  MoveC 5273 to (-170.79, 260.24, -44.5) mm, rotated rx -180 ry 0 rz 0.01 deg; joints [38.208, -42.51, 99.953, -137.192, 65.567, 159.929] to (-173.38, 259.8, -44.5) mm, rotated rx -180 ry 0 rz 0.01 deg; joints [38.136, -42.43, 99.783, -137.238, 65.475, 159.893]
  MoveC 5274 to (-175.99, 259.57, -44.5) mm, rotated rx 180 ry 0 rz 0.01 deg; joints [38.069, -42.344, 99.599, -137.276, 65.378, 159.849] to (-178.62, 259.49, -44.5) mm, rotated rx 180 ry 0 rz 0.01 deg; joints [38.007, -42.253, 99.403, -137.307, 65.279, 159.798]
  MoveL 5275 to (-216.35, 259.58, -44.5) mm, rotated rx 180 ry 0 rz 0.01 deg; joints [37.165, -40.878, 96.467, -137.67, 63.812, 159.01]
  MoveC 5276 to (-223.68, 260.93, -44.5) mm, rotated rx 180 ry 0 rz 0.01 deg; joints [37.043, -40.567, 95.803, -137.677, 63.505, 158.802] to (-230.83, 263.03, -44.5) mm, rotated rx 180 ry 0 rz 0.01 deg; joints [36.949, -40.24, 95.104, -137.649, 63.193, 158.566]
  MoveC 5277 to (-237.52, 266.44, -44.5) mm, rotated rx -180 ry 0 rz 0.01 deg; joints [36.902, -39.891, 94.357, -137.561, 62.881, 158.288] to (-243.08, 271.47, -44.5) mm, rotated rx -180 ry 0 rz 0.01 deg; joints [36.926, -39.537, 93.597, -137.394, 62.592, 157.967]
  MoveC 5278 to (-246.21, 275.5, -44.5) mm, rotated rx 180 ry 0 rz 0.01 deg; joints [36.974, -39.303, 93.093, -137.25, 62.413, 157.738] to (-248.99, 279.78, -44.5) mm, rotated rx 180 ry 0 rz 0.01 deg; joints [37.036, -39.073, 92.601, -137.092, 62.245, 157.506]
  MoveC 5279 to (-251.23, 284.38, -44.5) mm, rotated rx 180 ry 0 rz 0.01 deg; joints [37.118, -38.854, 92.13, -136.916, 62.094, 157.271] to (-252.73, 289.26, -44.5) mm, rotated rx -180 ry 0 rz 0.01 deg; joints [37.224, -38.654, 91.699, -136.724, 61.969, 157.04]
  MoveC 5280 to (-253.82, 296.03, -44.5) mm, rotated rx -180 ry 0 rz 0.01 deg; joints [37.39, -38.415, 91.182, -136.45, 61.836, 156.741] to (-254.09, 302.88, -44.5) mm, rotated rx 180 ry 0 rz 0.01 deg; joints [37.576, -38.202, 90.723, -136.168, 61.736, 156.455]
  MoveC 5281 to (-253.11, 309.7, -44.5) mm, rotated rx -180 ry 0 rz 0.01 deg; joints [37.786, -38.038, 90.366, -135.879, 61.686, 156.199] to (-250.53, 316.09, -44.5) mm, rotated rx -180 ry 0 rz 0.01 deg; joints [38.018, -37.948, 90.167, -135.6, 61.707, 155.997]
  MoveC 5282 to (-249.34, 318.22, -44.5) mm, rotated rx -180 ry 0 rz 0.01 deg; joints [38.102, -37.931, 90.127, -135.505, 61.727, 155.937] to (-248.13, 320.34, -44.5) mm, rotated rx 180 ry 0 rz 0.01 deg; joints [38.187, -37.915, 90.089, -135.41, 61.748, 155.878]
  MoveL 5283 to (-247.97, 320.95, -44.33) mm, rotated rx 180 ry 0 rz 0.01 deg; joints [38.207, -37.911, 90.064, -135.382, 61.741, 155.851]
  MoveL 5284 to (-248.05, 321.41, -43.87) mm, rotated rx -180 ry 0 rz 0.01 deg; joints [38.217, -37.915, 90.03, -135.356, 61.718, 155.815]
  MoveL 5285 to (-248.12, 321.56, -43.23) mm, rotated rx 180 ry 0 rz 0.01 deg; joints [38.22, -37.938, 90.017, -135.34, 61.694, 155.785]
  Set speed (500.0 mm/s)
  MoveL 5286 to (-248.12, 321.56, 11) mm, rotated rx -180 ry 0 rz 0.01 deg; joints [38.197, -40.432, 90.187, -134.447, 60.044, 153.913]
  Set speed (500.0 mm/s)
  MoveL 5287 to (-399.69, 339.08, 11) mm, rotated rx 180 ry 0 rz 0.01 deg; joints [35.607, -32.97, 75.014, -133.485, 53.388, 148.774]
  Set speed (100.0 mm/s)
  MoveL 5288 to (-399.69, 339.08, -28.23) mm, rotated rx -180 ry 0 rz 0.01 deg; joints [35.623, -31.334, 74.905, -134.27, 54.456, 150.126]
  MoveL 5289 to (-399.69, 339.08, -28.33) mm, rotated rx -180 ry 0 rz 0.01 deg; joints [35.623, -31.33, 74.904, -134.272, 54.458, 150.13]
  MoveL 5290 to (-399.83, 339.05, -28.81) mm, rotated rx -180 ry 0 rz 0.01 deg; joints [35.62, -31.303, 74.89, -134.281, 54.465, 150.142]
  MoveL 5291 to (-400.13, 338.98, -29.2) mm, rotated rx -180 ry 0 rz 0.01 deg; joints [35.613, -31.274, 74.862, -134.289, 54.462, 150.148]
  MoveL 5292 to (-400.55, 338.85, -29.44) mm, rotated rx -180 ry 0 rz 0.01 deg; joints [35.602, -31.247, 74.827, -134.297, 54.45, 150.148]
  MoveL 5293 to (-400.6, 338.83, -29.46) mm, rotated rx -180 ry 0 rz 0.01 deg; joints [35.6, -31.245, 74.824, -134.298, 54.449, 150.148]
  MoveL 5294 to (-400.86, 338.72, -29.5) mm, rotated rx 180 ry 0 rz 0.01 deg; joints [35.593, -31.234, 74.805, -134.302, 54.439, 150.145]
  MoveL 5295 to (-401.28, 338.49, -29.52) mm, rotated rx 180 ry 0 rz 0.01 deg; joints [35.579, -31.22, 74.778, -134.31, 54.423, 150.143]
  MoveL 5296 to (-401.4, 338.42, -29.52) mm, rotated rx 180 ry 0 rz 0.01 deg; joints [35.574, -31.216, 74.771, -134.313, 54.418, 150.142]
  MoveL 5297 to (-402.84, 337.05, -29.59) mm, rotated rx 180 ry 0 rz 0.01 deg; joints [35.511, -31.189, 74.722, -134.368, 54.371, 150.163]
  MoveL 5298 to (-402.87, 337.02, -29.59) mm, rotated rx -180 ry 0 rz 0.01 deg; joints [35.51, -31.189, 74.722, -134.37, 54.37, 150.164]
  MoveL 5299 to (-403.75, 334.43, -29.69) mm, rotated rx -180 ry 0 rz 0.01 deg; joints [35.425, -31.231, 74.821, -134.488, 54.366, 150.266]
  MoveL 5300 to (-403.78, 333.95, -29.71) mm, rotated rx -180 ry 0 rz 0.01 deg; joints [35.412, -31.246, 74.854, -134.511, 54.372, 150.29]
  MoveL 5301 to (-403.79, 333.65, -29.72) mm, rotated rx -180 ry 0 rz 0.01 deg; joints [35.404, -31.255, 74.874, -134.525, 54.375, 150.305]
  MoveL 5302 to (-403.79, 333.05, -29.74) mm, rotated rx -180 ry 0 rz 0.01 deg; joints [35.388, -31.276, 74.919, -134.554, 54.384, 150.336]
  MoveL 5303 to (-401.25, 328.08, -29.94) mm, rotated rx -180 ry 0 rz 0.01 deg; joints [35.304, -31.566, 75.542, -134.812, 54.575, 150.679]
  MoveL 5304 to (-395.74, 327.2, -30.14) mm, rotated rx -180 ry 0 rz 0.01 deg; joints [35.385, -31.86, 76.168, -134.893, 54.85, 150.918]
  MoveL 5305 to (-391.79, 331.15, -30.35) mm, rotated rx -180 ry 0 rz 0.01 deg; joints [35.564, -31.91, 76.283, -134.736, 54.987, 150.863]
  MoveL 5306 to (-392.66, 336.66, -30.55) mm, rotated rx -180 ry 0 rz 0.01 deg; joints [35.694, -31.668, 75.792, -134.476, 54.878, 150.567]
  MoveL 5307 to (-397.64, 339.2, -30.75) mm, rotated rx -180 ry 0 rz 0.01 deg; joints [35.666, -31.325, 75.096, -134.327, 54.617, 150.275]
  MoveL 5308 to (-398.51, 339.2, -30.78) mm, rotated rx -180 ry 0 rz 0.01 deg; joints [35.65, -31.28, 75.006, -134.321, 54.577, 150.246]
  MoveL 5309 to (-399.34, 339.13, -30.81) mm, rotated rx 180 ry 0 rz 0.01 deg; joints [35.633, -31.24, 74.926, -134.319, 54.54, 150.221]
  MoveL 5310 to (-399.69, 339.08, -30.82) mm, rotated rx -180 ry 0 rz 0.01 deg; joints [35.624, -31.223, 74.893, -134.319, 54.525, 150.212]
  MoveL 5311 to (-400.55, 338.85, -30.85) mm, rotated rx -180 ry 0 rz 0.01 deg; joints [35.602, -31.187, 74.821, -134.324, 54.488, 150.194]
  MoveL 5312 to (-400.6, 338.83, -30.85) mm, rotated rx -180 ry 0 rz 0.01 deg; joints [35.601, -31.185, 74.818, -134.324, 54.486, 150.194]
  MoveL 5313 to (-401.28, 338.49, -30.88) mm, rotated rx -180 ry 0 rz 0.01 deg; joints [35.579, -31.162, 74.772, -134.336, 54.459, 150.188]
  MoveL 5314 to (-401.4, 338.42, -30.89) mm, rotated rx -180 ry 0 rz 0.01 deg; joints [35.575, -31.158, 74.764, -134.339, 54.455, 150.187]
  MoveL 5315 to (-402.84, 337.05, -30.96) mm, rotated rx -180 ry 0 rz 0.01 deg; joints [35.512, -31.131, 74.716, -134.394, 54.407, 150.208]
  MoveL 5316 to (-402.87, 337.02, -30.96) mm, rotated rx -180 ry 0 rz 0.01 deg; joints [35.511, -31.131, 74.716, -134.395, 54.407, 150.209]
  MoveL 5317 to (-403.75, 334.43, -31.05) mm, rotated rx 180 ry 0 rz 0.01 deg; joints [35.426, -31.173, 74.814, -134.514, 54.402, 150.311]
  MoveL 5318 to (-403.78, 333.95, -31.07) mm, rotated rx -180 ry 0 rz 0.01 deg; joints [35.413, -31.188, 74.847, -134.537, 54.408, 150.335]
  MoveL 5319 to (-403.79, 333.65, -31.08) mm, rotated rx 180 ry 0 rz 0.01 deg; joints [35.405, -31.197, 74.868, -134.551, 54.412, 150.35]
  MoveL 5320 to (-403.79, 333.05, -31.1) mm, rotated rx 180 ry 0 rz 0.01 deg; joints [35.389, -31.217, 74.912, -134.58, 54.421, 150.381]
  MoveL 5321 to (-401.25, 328.08, -31.3) mm, rotated rx -180 ry 0 rz 0.01 deg; joints [35.305, -31.508, 75.536, -134.837, 54.612, 150.724]
  MoveL 5322 to (-395.74, 327.2, -31.51) mm, rotated rx 180 ry 0 rz 0.01 deg; joints [35.386, -31.801, 76.162, -134.918, 54.888, 150.962]
  MoveL 5323 to (-391.79, 331.15, -31.71) mm, rotated rx 180 ry 0 rz 0.01 deg; joints [35.565, -31.851, 76.276, -134.762, 55.024, 150.908]
  MoveL 5324 to (-392.66, 336.66, -31.91) mm, rotated rx 180 ry 0 rz 0.01 deg; joints [35.694, -31.609, 75.785, -134.502, 54.915, 150.612]
  MoveL 5325 to (-397.64, 339.2, -32.11) mm, rotated rx -180 ry 0 rz 0.01 deg; joints [35.667, -31.266, 75.089, -134.352, 54.654, 150.32]
  MoveL 5326 to (-398.51, 339.2, -32.14) mm, rotated rx -180 ry 0 rz 0.01 deg; joints [35.651, -31.222, 75, -134.347, 54.614, 150.291]
  MoveL 5327 to (-399.34, 339.13, -32.17) mm, rotated rx -180 ry 0 rz 0.01 deg; joints [35.633, -31.181, 74.919, -134.344, 54.577, 150.266]
  MoveL 5328 to (-399.69, 339.08, -32.19) mm, rotated rx 180 ry 0 rz 0.01 deg; joints [35.625, -31.165, 74.886, -134.345, 54.561, 150.257]
  MoveL 5329 to (-400.55, 338.85, -32.22) mm, rotated rx 180 ry 0 rz 0.01 deg; joints [35.603, -31.129, 74.814, -134.35, 54.525, 150.239]
  MoveL 5330 to (-400.6, 338.83, -32.22) mm, rotated rx -180 ry 0 rz 0.01 deg; joints [35.602, -31.127, 74.811, -134.35, 54.523, 150.239]
  MoveL 5331 to (-401.28, 338.49, -32.25) mm, rotated rx 180 ry 0 rz 0.01 deg; joints [35.58, -31.104, 74.765, -134.362, 54.496, 150.233]
  MoveL 5332 to (-401.4, 338.42, -32.25) mm, rotated rx -180 ry 0 rz 0.01 deg; joints [35.575, -31.1, 74.758, -134.364, 54.491, 150.232]
  MoveL 5333 to (-402.84, 337.05, -32.32) mm, rotated rx -180 ry 0 rz 0.01 deg; joints [35.513, -31.073, 74.709, -134.42, 54.444, 150.253]
  MoveL 5334 to (-402.87, 337.02, -32.32) mm, rotated rx -180 ry 0 rz 0.01 deg; joints [35.511, -31.073, 74.709, -134.421, 54.443, 150.254]
  MoveL 5335 to (-403.75, 334.43, -32.42) mm, rotated rx -180 ry 0 rz 0.01 deg; joints [35.426, -31.115, 74.808, -134.539, 54.439, 150.356]
  MoveL 5336 to (-403.78, 333.95, -32.44) mm, rotated rx -180 ry 0 rz 0.01 deg; joints [35.413, -31.13, 74.841, -134.562, 54.445, 150.38]
  MoveL 5337 to (-403.79, 333.65, -32.45) mm, rotated rx -180 ry 0 rz 0.01 deg; joints [35.405, -31.139, 74.861, -134.576, 54.449, 150.395]
  MoveL 5338 to (-403.79, 333.05, -32.47) mm, rotated rx -180 ry 0 rz 0.01 deg; joints [35.389, -31.159, 74.906, -134.605, 54.457, 150.426]
  MoveL 5339 to (-401.25, 328.08, -32.67) mm, rotated rx -180 ry 0 rz 0.01 deg; joints [35.306, -31.449, 75.529, -134.863, 54.649, 150.769]
  MoveL 5340 to (-395.74, 327.2, -32.87) mm, rotated rx 180 ry 0 rz 0.01 deg; joints [35.386, -31.743, 76.155, -134.944, 54.925, 151.007]
  MoveL 5341 to (-391.79, 331.15, -33.07) mm, rotated rx -180 ry 0 rz 0.01 deg; joints [35.565, -31.793, 76.27, -134.787, 55.061, 150.953]
  MoveL 5342 to (-392.66, 336.66, -33.28) mm, rotated rx -180 ry 0 rz 0.01 deg; joints [35.695, -31.551, 75.779, -134.527, 54.952, 150.657]
  MoveL 5343 to (-397.64, 339.2, -33.48) mm, rotated rx -180 ry 0 rz 0.01 deg; joints [35.668, -31.208, 75.083, -134.378, 54.69, 150.365]
  MoveL 5344 to (-398.51, 339.2, -33.51) mm, rotated rx -180 ry 0 rz 0.01 deg; joints [35.651, -31.163, 74.993, -134.372, 54.65, 150.336]
  MoveL 5345 to (-399.34, 339.13, -33.54) mm, rotated rx -180 ry 0 rz 0.01 deg; joints [35.634, -31.123, 74.912, -134.37, 54.613, 150.311]
  MoveL 5346 to (-399.69, 339.08, -33.55) mm, rotated rx -180 ry 0 rz 0.01 deg; joints [35.626, -31.107, 74.88, -134.37, 54.597, 150.302]
  MoveL 5347 to (-400.55, 338.85, -33.58) mm, rotated rx -180 ry 0 rz 0.01 deg; joints [35.603, -31.071, 74.807, -134.375, 54.561, 150.284]
  MoveL 5348 to (-400.6, 338.83, -33.58) mm, rotated rx -180 ry 0 rz 0.01 deg; joints [35.602, -31.069, 74.804, -134.376, 54.559, 150.284]
  MoveL 5349 to (-401.28, 338.49, -33.61) mm, rotated rx -180 ry 0 rz 0.01 deg; joints [35.58, -31.045, 74.758, -134.387, 54.532, 150.278]
  MoveL 5350 to (-401.4, 338.42, -33.62) mm, rotated rx -180 ry 0 rz 0.01 deg; joints [35.576, -31.042, 74.751, -134.39, 54.527, 150.277]
  MoveL 5351 to (-402.84, 337.05, -33.69) mm, rotated rx 180 ry 0 rz 0.01 deg; joints [35.513, -31.015, 74.703, -134.445, 54.48, 150.298]
  MoveL 5352 to (-402.87, 337.02, -33.69) mm, rotated rx -180 ry 0 rz 0.01 deg; joints [35.512, -31.015, 74.703, -134.447, 54.479, 150.299]
  MoveL 5353 to (-403.75, 334.43, -33.78) mm, rotated rx -180 ry 0 rz 0.01 deg; joints [35.427, -31.056, 74.801, -134.565, 54.475, 150.401]
  MoveL 5354 to (-403.78, 333.95, -33.8) mm, rotated rx 180 ry 0 rz 0.01 deg; joints [35.414, -31.071, 74.834, -134.588, 54.481, 150.425]
  MoveL 5355 to (-403.79, 333.65, -33.81) mm, rotated rx -180 ry 0 rz 0.01 deg; joints [35.406, -31.081, 74.855, -134.602, 54.485, 150.44]
  MoveL 5356 to (-403.79, 333.05, -33.83) mm, rotated rx -180 ry 0 rz 0.01 deg; joints [35.39, -31.101, 74.899, -134.631, 54.494, 150.471]
  MoveL 5357 to (-401.25, 328.08, -34.03) mm, rotated rx 180 ry 0 rz 0.01 deg; joints [35.306, -31.391, 75.523, -134.888, 54.686, 150.814]
  MoveL 5358 to (-395.74, 327.2, -34.24) mm, rotated rx -180 ry 0 rz 0.01 deg; joints [35.387, -31.684, 76.148, -134.969, 54.962, 151.052]
  MoveL 5359 to (-391.79, 331.15, -34.44) mm, rotated rx -180 ry 0 rz 0.01 deg; joints [35.566, -31.734, 76.263, -134.812, 55.098, 150.998]
  MoveL 5360 to (-392.66, 336.66, -34.64) mm, rotated rx -180 ry 0 rz 0.01 deg; joints [35.695, -31.492, 75.772, -134.552, 54.988, 150.702]
  MoveL 5361 to (-397.64, 339.2, -34.84) mm, rotated rx -180 ry 0 rz 0.01 deg; joints [35.668, -31.149, 75.076, -134.403, 54.727, 150.41]
  MoveL 5362 to (-398.51, 339.2, -34.87) mm, rotated rx 180 ry 0 rz 0.01 deg; joints [35.652, -31.105, 74.986, -134.398, 54.687, 150.381]
  MoveL 5363 to (-399.34, 339.13, -34.9) mm, rotated rx -180 ry 0 rz 0.01 deg; joints [35.634, -31.065, 74.905, -134.395, 54.649, 150.356]
  MoveL 5364 to (-399.69, 339.08, -34.92) mm, rotated rx -180 ry 0 rz 0.01 deg; joints [35.626, -31.048, 74.873, -134.396, 54.634, 150.347]
  MoveL 5365 to (-400.55, 338.85, -34.95) mm, rotated rx -180 ry 0 rz 0.01 deg; joints [35.604, -31.012, 74.801, -134.401, 54.597, 150.329]
  MoveL 5366 to (-400.6, 338.83, -34.95) mm, rotated rx -180 ry 0 rz 0.01 deg; joints [35.603, -31.011, 74.797, -134.401, 54.595, 150.329]
  MoveL 5367 to (-401.28, 338.49, -34.97) mm, rotated rx 180 ry 0 rz 0.01 deg; joints [35.581, -30.987, 74.751, -134.413, 54.568, 150.322]
  MoveL 5368 to (-401.4, 338.42, -34.98) mm, rotated rx -180 ry 0 rz 0.01 deg; joints [35.577, -30.983, 74.744, -134.416, 54.564, 150.322]
  MoveL 5369 to (-402.84, 337.05, -35.05) mm, rotated rx -180 ry 0 rz 0.01 deg; joints [35.514, -30.956, 74.696, -134.471, 54.516, 150.342]
  MoveL 5370 to (-402.87, 337.02, -35.05) mm, rotated rx -180 ry 0 rz 0.01 deg; joints [35.512, -30.956, 74.696, -134.472, 54.516, 150.343]
  MoveL 5371 to (-403.75, 334.43, -35.15) mm, rotated rx -180 ry 0 rz 0.01 deg; joints [35.428, -30.998, 74.794, -134.59, 54.512, 150.445]
  MoveL 5372 to (-403.78, 333.95, -35.16) mm, rotated rx 180 ry 0 rz 0.01 deg; joints [35.414, -31.013, 74.827, -134.613, 54.518, 150.469]
  MoveL 5373 to (-403.79, 333.65, -35.18) mm, rotated rx 180 ry 0 rz 0.01 deg; joints [35.406, -31.022, 74.848, -134.628, 54.521, 150.484]
  MoveL 5374 to (-403.79, 333.05, -35.2) mm, rotated rx -180 ry 0 rz 0.01 deg; joints [35.391, -31.042, 74.892, -134.657, 54.53, 150.515]
  MoveL 5375 to (-401.25, 328.08, -35.4) mm, rotated rx -180 ry 0 rz 0.01 deg; joints [35.307, -31.332, 75.516, -134.913, 54.723, 150.858]
  MoveL 5376 to (-395.74, 327.2, -35.6) mm, rotated rx -180 ry 0 rz 0.01 deg; joints [35.387, -31.625, 76.141, -134.994, 54.999, 151.096]
  MoveL 5377 to (-391.79, 331.15, -35.8) mm, rotated rx -180 ry 0 rz 0.01 deg; joints [35.567, -31.675, 76.256, -134.837, 55.135, 151.042]
  MoveL 5378 to (-392.66, 336.66, -36.01) mm, rotated rx -180 ry 0 rz 0.01 deg; joints [35.696, -31.434, 75.765, -134.577, 55.025, 150.747]
  MoveL 5379 to (-397.64, 339.2, -36.21) mm, rotated rx 180 ry 0 rz 0.01 deg; joints [35.669, -31.091, 75.069, -134.429, 54.763, 150.455]
  MoveL 5380 to (-398.51, 339.2, -36.24) mm, rotated rx -180 ry 0 rz 0.01 deg; joints [35.652, -31.046, 74.979, -134.423, 54.723, 150.426]
  MoveL 5381 to (-399.34, 339.13, -36.27) mm, rotated rx 180 ry 0 rz 0.01 deg; joints [35.635, -31.006, 74.898, -134.421, 54.686, 150.401]
  MoveL 5382 to (-399.69, 339.08, -36.28) mm, rotated rx 180 ry 0 rz 0.01 deg; joints [35.627, -30.99, 74.866, -134.421, 54.67, 150.392]
  MoveL 5383 to (-400.55, 338.85, -36.31) mm, rotated rx 180 ry 0 rz 0.01 deg; joints [35.605, -30.954, 74.793, -134.426, 54.633, 150.374]
  MoveL 5384 to (-400.6, 338.83, -36.31) mm, rotated rx 180 ry 0 rz 0.01 deg; joints [35.603, -30.952, 74.79, -134.427, 54.632, 150.373]
  MoveL 5385 to (-401.28, 338.49, -36.34) mm, rotated rx -180 ry 0 rz 0.01 deg; joints [35.582, -30.929, 74.744, -134.438, 54.605, 150.367]
  MoveL 5386 to (-401.4, 338.42, -36.34) mm, rotated rx -180 ry 0 rz 0.01 deg; joints [35.577, -30.925, 74.737, -134.441, 54.6, 150.367]
  MoveL 5387 to (-402.84, 337.05, -36.41) mm, rotated rx -180 ry 0 rz 0.01 deg; joints [35.514, -30.898, 74.689, -134.496, 54.553, 150.387]
  MoveL 5388 to (-402.87, 337.02, -36.42) mm, rotated rx -180 ry 0 rz 0.01 deg; joints [35.513, -30.898, 74.689, -134.498, 54.552, 150.388]
  MoveL 5389 to (-403.75, 334.43, -36.51) mm, rotated rx -180 ry 0 rz 0.01 deg; joints [35.428, -30.94, 74.787, -134.616, 54.548, 150.49]
  MoveL 5390 to (-403.78, 333.95, -36.53) mm, rotated rx -180 ry 0 rz 0.01 deg; joints [35.415, -30.954, 74.82, -134.639, 54.554, 150.514]
  MoveL 5391 to (-403.79, 333.65, -36.54) mm, rotated rx -180 ry 0 rz 0.01 deg; joints [35.407, -30.964, 74.841, -134.653, 54.558, 150.529]
  MoveL 5392 to (-403.79, 333.05, -36.56) mm, rotated rx -180 ry 0 rz 0.01 deg; joints [35.391, -30.984, 74.885, -134.682, 54.567, 150.56]
  MoveL 5393 to (-401.25, 328.08, -36.76) mm, rotated rx 180 ry 0 rz 0.01 deg; joints [35.307, -31.273, 75.509, -134.938, 54.759, 150.902]
  MoveL 5394 to (-395.74, 327.2, -36.97) mm, rotated rx -180 ry 0 rz 0.01 deg; joints [35.388, -31.566, 76.134, -135.019, 55.036, 151.14]
  MoveL 5395 to (-391.79, 331.15, -37.17) mm, rotated rx -180 ry 0 rz 0.01 deg; joints [35.567, -31.616, 76.249, -134.862, 55.172, 151.086]
  MoveL 5396 to (-392.66, 336.66, -37.37) mm, rotated rx 180 ry 0 rz 0.01 deg; joints [35.697, -31.375, 75.758, -134.603, 55.061, 150.791]
  MoveL 5397 to (-397.64, 339.2, -37.57) mm, rotated rx -180 ry 0 rz 0.01 deg; joints [35.669, -31.032, 75.061, -134.454, 54.799, 150.499]
  MoveL 5398 to (-398.51, 339.2, -37.6) mm, rotated rx 180 ry 0 rz 0.01 deg; joints [35.653, -30.988, 74.972, -134.448, 54.759, 150.47]
  MoveL 5399 to (-399.34, 339.13, -37.63) mm, rotated rx -180 ry 0 rz 0.01 deg; joints [35.636, -30.948, 74.891, -134.446, 54.722, 150.445]
  MoveL 5400 to (-399.69, 339.08, -37.64) mm, rotated rx 180 ry 0 rz 0.01 deg; joints [35.627, -30.931, 74.858, -134.447, 54.706, 150.436]
  MoveL 5401 to (-400.55, 338.85, -37.68) mm, rotated rx 180 ry 0 rz 0.01 deg; joints [35.605, -30.895, 74.786, -134.452, 54.67, 150.418]
  MoveL 5402 to (-400.6, 338.83, -37.68) mm, rotated rx -180 ry 0 rz 0.01 deg; joints [35.604, -30.894, 74.783, -134.452, 54.668, 150.418]
  MoveL 5403 to (-401.28, 338.49, -37.7) mm, rotated rx 180 ry 0 rz 0.01 deg; joints [35.582, -30.87, 74.737, -134.464, 54.641, 150.411]
  MoveL 5404 to (-401.4, 338.42, -37.71) mm, rotated rx -180 ry 0 rz 0.01 deg; joints [35.578, -30.866, 74.73, -134.466, 54.636, 150.411]
  MoveL 5405 to (-402.84, 337.05, -37.78) mm, rotated rx -180 ry 0 rz 0.01 deg; joints [35.515, -30.839, 74.681, -134.522, 54.589, 150.431]
  MoveL 5406 to (-402.87, 337.02, -37.78) mm, rotated rx -180 ry 0 rz 0.01 deg; joints [35.514, -30.839, 74.681, -134.523, 54.588, 150.432]
  MoveL 5407 to (-403.75, 334.43, -37.88) mm, rotated rx -180 ry 0 rz 0.01 deg; joints [35.429, -30.881, 74.78, -134.641, 54.584, 150.534]
  MoveL 5408 to (-403.78, 333.95, -37.89) mm, rotated rx -180 ry 0 rz 0.01 deg; joints [35.416, -30.896, 74.813, -134.664, 54.59, 150.558]
  MoveL 5409 to (-403.79, 333.65, -37.9) mm, rotated rx 180 ry 0 rz 0.01 deg; joints [35.408, -30.905, 74.833, -134.678, 54.594, 150.573]
  MoveL 5410 to (-403.79, 333.05, -37.93) mm, rotated rx -180 ry 0 rz 0.01 deg; joints [35.392, -30.925, 74.878, -134.707, 54.603, 150.604]
  MoveL 5411 to (-401.25, 328.08, -38.13) mm, rotated rx -180 ry 0 rz 0.01 deg; joints [35.308, -31.215, 75.501, -134.964, 54.796, 150.947]
  MoveL 5412 to (-395.74, 327.2, -38.33) mm, rotated rx -180 ry 0 rz 0.01 deg; joints [35.389, -31.507, 76.127, -135.044, 55.072, 151.185]
  MoveL 5413 to (-391.79, 331.15, -38.53) mm, rotated rx 180 ry 0 rz 0.01 deg; joints [35.568, -31.557, 76.242, -134.887, 55.209, 151.131]
  MoveL 5414 to (-392.66, 336.66, -38.73) mm, rotated rx 180 ry 0 rz 0.01 deg; joints [35.697, -31.316, 75.751, -134.628, 55.098, 150.835]
  MoveL 5415 to (-397.64, 339.2, -38.94) mm, rotated rx 180 ry 0 rz 0.01 deg; joints [35.67, -30.974, 75.054, -134.479, 54.835, 150.544]
  MoveL 5416 to (-398.51, 339.2, -38.97) mm, rotated rx -180 ry 0 rz 0.01 deg; joints [35.654, -30.929, 74.964, -134.474, 54.795, 150.514]
  MoveL 5417 to (-399.34, 339.13, -39) mm, rotated rx 180 ry 0 rz 0.01 deg; joints [35.636, -30.889, 74.884, -134.471, 54.758, 150.49]
  MoveL 5418 to (-399.69, 339.08, -39.01) mm, rotated rx -180 ry 0 rz 0.01 deg; joints [35.628, -30.873, 74.851, -134.472, 54.742, 150.48]
  MoveL 5419 to (-400.55, 338.85, -39.04) mm, rotated rx -180 ry 0 rz 0.01 deg; joints [35.606, -30.837, 74.779, -134.477, 54.706, 150.463]
  MoveL 5420 to (-400.6, 338.83, -39.04) mm, rotated rx 180 ry 0 rz 0.01 deg; joints [35.605, -30.835, 74.776, -134.477, 54.704, 150.462]
  MoveL 5421 to (-401.28, 338.49, -39.07) mm, rotated rx 180 ry 0 rz 0.01 deg; joints [35.583, -30.811, 74.73, -134.489, 54.677, 150.456]
  MoveL 5422 to (-401.4, 338.42, -39.07) mm, rotated rx 180 ry 0 rz 0.01 deg; joints [35.578, -30.808, 74.722, -134.492, 54.672, 150.456]
  MoveL 5423 to (-402.84, 337.05, -39.14) mm, rotated rx 180 ry 0 rz 0.01 deg; joints [35.516, -30.781, 74.674, -134.547, 54.625, 150.476]
  MoveL 5424 to (-402.87, 337.02, -39.14) mm, rotated rx 180 ry 0 rz 0.01 deg; joints [35.514, -30.781, 74.674, -134.549, 54.624, 150.477]
  MoveL 5425 to (-403.75, 334.43, -39.24) mm, rotated rx 180 ry 0 rz 0.01 deg; joints [35.429, -30.822, 74.772, -134.666, 54.621, 150.579]
  MoveL 5426 to (-403.78, 333.95, -39.26) mm, rotated rx 180 ry 0 rz 0.01 deg; joints [35.416, -30.837, 74.805, -134.689, 54.627, 150.603]
  MoveL 5427 to (-403.79, 333.65, -39.27) mm, rotated rx 180 ry 0 rz 0.01 deg; joints [35.408, -30.847, 74.826, -134.704, 54.631, 150.617]
  MoveL 5428 to (-403.79, 333.05, -39.29) mm, rotated rx 180 ry 0 rz 0.01 deg; joints [35.392, -30.867, 74.87, -134.732, 54.639, 150.648]
  MoveL 5429 to (-401.25, 328.08, -39.49) mm, rotated rx 180 ry 0 rz 0.01 deg; joints [35.308, -31.156, 75.494, -134.989, 54.833, 150.991]
  MoveL 5430 to (-395.74, 327.2, -39.69) mm, rotated rx 180 ry 0 rz 0.01 deg; joints [35.389, -31.448, 76.12, -135.069, 55.109, 151.229]
  MoveL 5431 to (-391.79, 331.15, -39.9) mm, rotated rx -180 ry 0 rz 0.01 deg; joints [35.568, -31.498, 76.234, -134.912, 55.245, 151.175]
  MoveL 5432 to (-392.66, 336.66, -40.1) mm, rotated rx -180 ry 0 rz 0.01 deg; joints [35.698, -31.257, 75.743, -134.652, 55.134, 150.88]
  MoveL 5433 to (-397.64, 339.2, -40.3) mm, rotated rx -180 ry 0 rz 0.01 deg; joints [35.67, -30.915, 75.046, -134.504, 54.872, 150.588]
  MoveL 5434 to (-398.51, 339.2, -40.33) mm, rotated rx -180 ry 0 rz 0.01 deg; joints [35.654, -30.871, 74.957, -134.499, 54.832, 150.559]
  MoveL 5435 to (-399.34, 339.13, -40.36) mm, rotated rx -180 ry 0 rz 0.01 deg; joints [35.637, -30.83, 74.876, -134.497, 54.794, 150.534]
  MoveL 5436 to (-399.69, 339.08, -40.37) mm, rotated rx 180 ry 0 rz 0.01 deg; joints [35.629, -30.814, 74.843, -134.497, 54.779, 150.525]
  MoveL 5437 to (-400.55, 338.85, -40.4) mm, rotated rx 180 ry 0 rz 0.01 deg; joints [35.606, -30.778, 74.771, -134.502, 54.742, 150.507]
  MoveL 5438 to (-400.6, 338.83, -40.41) mm, rotated rx 180 ry 0 rz 0.01 deg; joints [35.605, -30.776, 74.768, -134.503, 54.74, 150.506]
  MoveL 5439 to (-401.28, 338.49, -40.43) mm, rotated rx 180 ry 0 rz 0.01 deg; joints [35.583, -30.753, 74.722, -134.514, 54.713, 150.5]
  MoveL 5440 to (-401.4, 338.42, -40.44) mm, rotated rx -180 ry 0 rz 0.01 deg; joints [35.579, -30.749, 74.715, -134.517, 54.709, 150.5]
  MoveL 5441 to (-402.84, 337.05, -40.51) mm, rotated rx -180 ry 0 rz 0.01 deg; joints [35.516, -30.722, 74.666, -134.572, 54.661, 150.52]
  MoveL 5442 to (-402.87, 337.02, -40.51) mm, rotated rx -180 ry 0 rz 0.01 deg; joints [35.515, -30.722, 74.666, -134.574, 54.661, 150.521]
  MoveL 5443 to (-403.75, 334.43, -40.61) mm, rotated rx -180 ry 0 rz 0.01 deg; joints [35.43, -30.764, 74.765, -134.692, 54.657, 150.623]
  MoveL 5444 to (-403.78, 333.95, -40.62) mm, rotated rx -180 ry 0 rz 0.01 deg; joints [35.417, -30.779, 74.798, -134.715, 54.663, 150.647]
  MoveL 5445 to (-403.79, 333.65, -40.63) mm, rotated rx 180 ry 0 rz 0.01 deg; joints [35.409, -30.788, 74.818, -134.729, 54.667, 150.662]
  MoveL 5446 to (-403.79, 333.05, -40.65) mm, rotated rx -180 ry 0 rz 0.01 deg; joints [35.393, -30.808, 74.863, -134.758, 54.676, 150.693]
  MoveL 5447 to (-401.25, 328.08, -40.86) mm, rotated rx 180 ry 0 rz 0.01 deg; joints [35.309, -31.097, 75.486, -135.014, 54.869, 151.035]
  MoveL 5448 to (-395.74, 327.2, -41.06) mm, rotated rx 180 ry 0 rz 0.01 deg; joints [35.39, -31.389, 76.112, -135.093, 55.146, 151.273]
  MoveL 5449 to (-391.79, 331.15, -41.26) mm, rotated rx 180 ry 0 rz 0.01 deg; joints [35.569, -31.439, 76.227, -134.936, 55.282, 151.219]
  MoveL 5450 to (-392.66, 336.66, -41.46) mm, rotated rx -180 ry 0 rz 0.01 deg; joints [35.698, -31.198, 75.735, -134.677, 55.171, 150.924]
  MoveL 5451 to (-397.64, 339.2, -41.67) mm, rotated rx 180 ry 0 rz 0.01 deg; joints [35.671, -30.856, 75.039, -134.529, 54.908, 150.632]
  MoveL 5452 to (-398.51, 339.2, -41.7) mm, rotated rx -180 ry 0 rz 0.01 deg; joints [35.655, -30.812, 74.949, -134.524, 54.868, 150.603]
  MoveL 5453 to (-399.34, 339.13, -41.73) mm, rotated rx -180 ry 0 rz 0.01 deg; joints [35.637, -30.772, 74.868, -134.522, 54.83, 150.578]
  MoveL 5454 to (-399.69, 339.08, -41.74) mm, rotated rx -180 ry 0 rz 0.01 deg; joints [35.629, -30.755, 74.836, -134.522, 54.815, 150.569]
  MoveL 5455 to (-400.55, 338.85, -41.77) mm, rotated rx 180 ry 0 rz 0.01 deg; joints [35.607, -30.719, 74.764, -134.527, 54.778, 150.551]
  MoveL 5456 to (-400.6, 338.83, -41.77) mm, rotated rx -180 ry 0 rz 0.01 deg; joints [35.606, -30.718, 74.76, -134.528, 54.776, 150.551]
  MoveL 5457 to (-401.28, 338.49, -41.8) mm, rotated rx 180 ry 0 rz 0.01 deg; joints [35.584, -30.694, 74.714, -134.539, 54.749, 150.544]
  MoveL 5458 to (-401.4, 338.42, -41.8) mm, rotated rx -180 ry 0 rz 0.01 deg; joints [35.58, -30.69, 74.707, -134.542, 54.745, 150.544]
  MoveL 5459 to (-402.84, 337.05, -41.87) mm, rotated rx 180 ry 0 rz 0.01 deg; joints [35.517, -30.663, 74.659, -134.597, 54.697, 150.564]
  MoveL 5460 to (-402.87, 337.02, -41.87) mm, rotated rx 180 ry 0 rz 0.01 deg; joints [35.515, -30.663, 74.659, -134.599, 54.697, 150.565]
  MoveL 5461 to (-403.75, 334.43, -41.97) mm, rotated rx 180 ry 0 rz 0.01 deg; joints [35.431, -30.705, 74.757, -134.717, 54.693, 150.667]
  MoveL 5462 to (-403.78, 333.95, -41.99) mm, rotated rx -180 ry 0 rz 0.01 deg; joints [35.417, -30.72, 74.79, -134.74, 54.699, 150.691]
  MoveL 5463 to (-403.79, 333.65, -42) mm, rotated rx -180 ry 0 rz 0.01 deg; joints [35.409, -30.729, 74.811, -134.754, 54.703, 150.706]
  MoveL 5464 to (-403.79, 333.05, -42.02) mm, rotated rx -180 ry 0 rz 0.01 deg; joints [35.394, -30.749, 74.855, -134.783, 54.712, 150.737]
  MoveL 5465 to (-401.25, 328.08, -42.22) mm, rotated rx 180 ry 0 rz 0.01 deg; joints [35.31, -31.038, 75.478, -135.038, 54.906, 151.079]
  MoveL 5466 to (-395.74, 327.2, -42.42) mm, rotated rx -180 ry 0 rz 0.01 deg; joints [35.39, -31.33, 76.104, -135.118, 55.183, 151.317]
  MoveL 5467 to (-391.79, 331.15, -42.63) mm, rotated rx -180 ry 0 rz 0.01 deg; joints [35.57, -31.38, 76.219, -134.961, 55.319, 151.263]
  MoveL 5468 to (-392.66, 336.66, -42.83) mm, rotated rx 180 ry 0 rz 0.01 deg; joints [35.699, -31.139, 75.728, -134.702, 55.207, 150.968]
  MoveL 5469 to (-397.64, 339.2, -43.03) mm, rotated rx -180 ry 0 rz 0.01 deg; joints [35.672, -30.797, 75.031, -134.554, 54.944, 150.676]
  MoveL 5470 to (-398.51, 339.2, -43.06) mm, rotated rx -180 ry 0 rz 0.01 deg; joints [35.655, -30.753, 74.941, -134.549, 54.904, 150.647]
  MoveL 5471 to (-399.34, 339.13, -43.09) mm, rotated rx 180 ry 0 rz 0.01 deg; joints [35.638, -30.713, 74.86, -134.547, 54.866, 150.622]
  MoveL 5472 to (-399.69, 339.08, -43.1) mm, rotated rx 180 ry 0 rz 0.01 deg; joints [35.63, -30.696, 74.828, -134.547, 54.851, 150.613]
  MoveL 5473 to (-400.55, 338.85, -43.13) mm, rotated rx -180 ry 0 rz 0.01 deg; joints [35.608, -30.66, 74.756, -134.552, 54.814, 150.595]
  MoveL 5474 to (-400.6, 338.83, -43.14) mm, rotated rx -180 ry 0 rz 0.01 deg; joints [35.606, -30.659, 74.752, -134.553, 54.812, 150.595]
  MoveL 5475 to (-401.28, 338.49, -43.16) mm, rotated rx -180 ry 0 rz 0.01 deg; joints [35.584, -30.635, 74.706, -134.564, 54.785, 150.588]
  MoveL 5476 to (-401.4, 338.42, -43.17) mm, rotated rx 180 ry 0 rz 0.01 deg; joints [35.58, -30.632, 74.699, -134.567, 54.781, 150.588]
  MoveL 5477 to (-402.84, 337.05, -43.24) mm, rotated rx -180 ry 0 rz 0.01 deg; joints [35.517, -30.604, 74.651, -134.622, 54.733, 150.608]
  MoveL 5478 to (-402.87, 337.02, -43.24) mm, rotated rx -180 ry 0 rz 0.01 deg; joints [35.516, -30.604, 74.651, -134.624, 54.733, 150.609]
  MoveL 5479 to (-403.75, 334.43, -43.34) mm, rotated rx 180 ry 0 rz 0.01 deg; joints [35.431, -30.646, 74.749, -134.742, 54.729, 150.711]
  MoveL 5480 to (-403.78, 333.95, -43.35) mm, rotated rx -180 ry 0 rz 0.01 deg; joints [35.418, -30.661, 74.782, -134.765, 54.735, 150.735]
  MoveL 5481 to (-403.79, 333.65, -43.36) mm, rotated rx -180 ry 0 rz 0.01 deg; joints [35.41, -30.67, 74.803, -134.779, 54.739, 150.75]
  MoveL 5482 to (-403.79, 333.05, -43.38) mm, rotated rx -180 ry 0 rz 0.01 deg; joints [35.394, -30.69, 74.847, -134.808, 54.748, 150.78]
  MoveL 5483 to (-401.25, 328.08, -43.59) mm, rotated rx -180 ry 0 rz 0.01 deg; joints [35.31, -30.979, 75.471, -135.063, 54.942, 151.123]
  MoveL 5484 to (-395.74, 327.2, -43.79) mm, rotated rx -180 ry 0 rz 0.01 deg; joints [35.391, -31.271, 76.097, -135.143, 55.219, 151.36]
  MoveL 5485 to (-391.79, 331.15, -43.99) mm, rotated rx -180 ry 0 rz 0.01 deg; joints [35.57, -31.32, 76.211, -134.986, 55.355, 151.307]
  MoveL 5486 to (-392.66, 336.66, -44.19) mm, rotated rx -180 ry 0 rz 0.01 deg; joints [35.7, -31.08, 75.72, -134.727, 55.244, 151.012]
  MoveL 5487 to (-397.64, 339.2, -44.4) mm, rotated rx -180 ry 0 rz 0.01 deg; joints [35.672, -30.738, 75.023, -134.579, 54.98, 150.72]
  MoveL 5488 to (-398.51, 339.2, -44.43) mm, rotated rx -180 ry 0 rz 0.01 deg; joints [35.656, -30.694, 74.933, -134.574, 54.94, 150.691]
  MoveL 5489 to (-399.34, 339.13, -44.45) mm, rotated rx -180 ry 0 rz 0.01 deg; joints [35.639, -30.654, 74.852, -134.571, 54.902, 150.666]
  MoveL 5490 to (-399.69, 339.08, -44.47) mm, rotated rx -180 ry 0 rz 0.01 deg; joints [35.63, -30.638, 74.82, -134.572, 54.887, 150.657]
  MoveL 5491 to (-400.55, 338.85, -44.5) mm, rotated rx -180 ry 0 rz 0.01 deg; joints [35.608, -30.601, 74.748, -134.577, 54.85, 150.639]
  MoveL 5492 to (-400.6, 338.83, -44.5) mm, rotated rx -180 ry 0 rz 0.01 deg; joints [35.607, -30.6, 74.744, -134.578, 54.848, 150.639]
  MoveL 5493 to (-400.13, 339.01, -44.5) mm, rotated rx 180 ry 0 rz 0.01 deg; joints [35.62, -30.617, 74.779, -134.573, 54.868, 150.646]
  MoveL 5494 to (-398.92, 339.2, -44.5) mm, rotated rx 180 ry 0 rz 0.01 deg; joints [35.648, -30.67, 74.89, -134.572, 54.922, 150.679]
  MoveL 5495 to (-213.38, 339.2, -44.5) mm, rotated rx -180 ry 0 rz 0.01 deg; joints [39.469, -38.685, 91.691, -134.412, 62.886, 155.921]
  MoveL 5496 to (-213.56, 339.16, -44.5) mm, rotated rx 180 ry 0 rz 0.01 deg; joints [39.464, -38.68, 91.679, -134.415, 62.88, 155.919]
  MoveL 5497 to (-214.65, 338.88, -44.5) mm, rotated rx -180 ry 0 rz 0.01 deg; joints [39.432, -38.647, 91.61, -134.434, 62.84, 155.905]
  MoveL 5498 to (-215.28, 338.65, -44.5) mm, rotated rx 180 ry 0 rz 0.01 deg; joints [39.411, -38.63, 91.574, -134.448, 62.819, 155.9]
  MoveL 5499 to (-226.16, 333.38, -44.5) mm, rotated rx -180 ry 0 rz 0.01 deg; joints [39.025, -38.374, 91.041, -134.739, 62.458, 155.862]
  MoveL 5500 to (-226.67, 333.08, -44.5) mm, rotated rx -180 ry 0 rz 0.01 deg; joints [39.005, -38.364, 91.02, -134.754, 62.441, 155.862]
  MoveL 5501 to (-228.12, 332.03, -44.5) mm, rotated rx 180 ry 0 rz 0.01 deg; joints [38.945, -38.34, 90.971, -134.807, 62.397, 155.872]
  MoveL 5502 to (-228.46, 331.75, -44.5) mm, rotated rx 180 ry 0 rz 0.01 deg; joints [38.929, -38.335, 90.961, -134.821, 62.388, 155.875]
  MoveL 5503 to (-236.65, 324.01, -44.5) mm, rotated rx 180 ry 0 rz 0.01 deg; joints [38.538, -38.253, 90.798, -135.19, 62.162, 156.001]
  MoveL 5504 to (-236.97, 323.67, -44.5) mm, rotated rx -180 ry 0 rz 0.01 deg; joints [38.521, -38.251, 90.795, -135.207, 62.154, 156.008]
  MoveL 5505 to (-237.84, 322.58, -44.5) mm, rotated rx 180 ry 0 rz 0.01 deg; joints [38.472, -38.25, 90.794, -135.257, 62.133, 156.032]
  MoveL 5506 to (-238.12, 322.17, -44.5) mm, rotated rx 180 ry 0 rz 0.01 deg; joints [38.455, -38.251, 90.798, -135.275, 62.128, 156.042]
  MoveL 5507 to (-240.45, 318.18, -44.5) mm, rotated rx -180 ry 0 rz 0.01 deg; joints [38.294, -38.281, 90.866, -135.454, 62.087, 156.152]
  MoveL 5508 to (-240.48, 318.11, -44.5) mm, rotated rx 180 ry 0 rz 0.01 deg; joints [38.291, -38.281, 90.867, -135.457, 62.086, 156.153]
  MoveL 5509 to (-243.69, 312.31, -44.5) mm, rotated rx 180 ry 0 rz 0.01 deg; joints [38.061, -38.33, 90.978, -135.716, 62.033, 156.316]
  MoveL 5510 to (-243.88, 311.93, -44.5) mm, rotated rx -180 ry 0 rz 0.01 deg; joints [38.047, -38.334, 90.988, -135.733, 62.031, 156.327]
  MoveL 5511 to (-244.74, 309.75, -44.5) mm, rotated rx -180 ry 0 rz 0.01 deg; joints [37.968, -38.365, 91.057, -135.828, 62.024, 156.396]
  MoveL 5512 to (-244.95, 309.01, -44.5) mm, rotated rx -180 ry 0 rz 0.01 deg; joints [37.943, -38.379, 91.088, -135.86, 62.026, 156.422]
  MoveL 5513 to (-246.39, 299.58, -44.5) mm, rotated rx -180 ry 0 rz 0.01 deg; joints [37.649, -38.601, 91.572, -136.258, 62.091, 156.772]
  MoveL 5514 to (-246.42, 299.36, -44.5) mm, rotated rx -180 ry 0 rz 0.01 deg; joints [37.642, -38.607, 91.583, -136.268, 62.093, 156.78]
  MoveL 5515 to (-246.51, 298.27, -44.5) mm, rotated rx 180 ry 0 rz 0.01 deg; joints [37.61, -38.635, 91.645, -136.313, 62.103, 156.822]
  MoveC 5516 to (-246.51, 297.75, -44.5) mm, rotated rx -180 ry 0 rz 0.01 deg; joints [37.595, -38.65, 91.677, -136.334, 62.11, 156.843] to (-246.44, 297.24, -44.5) mm, rotated rx 180 ry 0 rz 0.01 deg; joints [37.583, -38.668, 91.716, -136.355, 62.12, 156.865]
  MoveL 5517 to (-245.04, 290.98, -44.5) mm, rotated rx 180 ry 0 rz 0.01 deg; joints [37.437, -38.904, 92.226, -136.604, 62.258, 157.15]
  MoveL 5518 to (-245.03, 290.91, -44.5) mm, rotated rx 180 ry 0 rz 0.01 deg; joints [37.435, -38.907, 92.231, -136.607, 62.259, 157.153]
  MoveL 5519 to (-244.07, 287.02, -44.5) mm, rotated rx 180 ry 0 rz 0.01 deg; joints [37.346, -39.056, 92.554, -136.761, 62.349, 157.331]
  MoveL 5520 to (-243.74, 286.17, -44.5) mm, rotated rx -180 ry 0 rz 0.01 deg; joints [37.329, -39.094, 92.635, -136.794, 62.373, 157.372]
  MoveL 5521 to (-241.01, 281.31, -44.5) mm, rotated rx 180 ry 0 rz 0.01 deg; joints [37.251, -39.338, 93.16, -136.975, 62.547, 157.627]
  MoveL 5522 to (-240.64, 280.78, -44.5) mm, rotated rx 180 ry 0 rz 0.01 deg; joints [37.244, -39.367, 93.223, -136.994, 62.568, 157.657]
  MoveL 5523 to (-237.07, 276.57, -44.5) mm, rotated rx 180 ry 0 rz 0.01 deg; joints [37.201, -39.624, 93.773, -137.142, 62.767, 157.903]
  MoveL 5524 to (-236.52, 276.04, -44.5) mm, rotated rx 180 ry 0 rz 0.01 deg; joints [37.198, -39.66, 93.851, -137.16, 62.796, 157.936]
  MoveL 5525 to (-230.7, 271.71, -44.5) mm, rotated rx 180 ry 0 rz 0.01 deg; joints [37.2, -40.003, 94.587, -137.293, 63.085, 158.234]
  MoveL 5526 to (-230.16, 271.37, -44.5) mm, rotated rx -180 ry 0 rz 0.01 deg; joints [37.203, -40.033, 94.651, -137.303, 63.111, 158.259]
  MoveL 5527 to (-227.13, 269.9, -44.5) mm, rotated rx -180 ry 0 rz 0.01 deg; joints [37.227, -40.189, 94.984, -137.339, 63.251, 158.382]
  MoveL 5528 to (-226.73, 269.74, -44.5) mm, rotated rx -180 ry 0 rz 0.01 deg; joints [37.23, -40.208, 95.025, -137.342, 63.268, 158.397]
  MoveL 5529 to (-222.87, 268.44, -44.5) mm, rotated rx -180 ry 0 rz 0.01 deg; joints [37.277, -40.39, 95.414, -137.364, 63.439, 158.532]
  MoveL 5530 to (-222.22, 268.29, -44.5) mm, rotated rx 180 ry 0 rz 0.01 deg; joints [37.287, -40.418, 95.474, -137.365, 63.466, 158.552]
  MoveL 5531 to (-215.33, 267.39, -44.5) mm, rotated rx -180 ry 0 rz 0.01 deg; joints [37.413, -40.701, 96.077, -137.343, 63.75, 158.735]
  MoveL 5532 to (-214.9, 267.36, -44.5) mm, rotated rx -180 ry 0 rz 0.01 deg; joints [37.422, -40.718, 96.113, -137.341, 63.768, 158.745]
  MoveL 5533 to (-178.62, 267.36, -44.5) mm, rotated rx 180 ry 0 rz 0.01 deg; joints [38.236, -42.039, 98.933, -136.992, 65.175, 159.505]
  MoveL 5534 to (-178.18, 267.39, -44.5) mm, rotated rx -180 ry 0 rz 0.01 deg; joints [38.247, -42.054, 98.964, -136.986, 65.192, 159.513]
  MoveL 5535 to (-171.29, 268.29, -44.5) mm, rotated rx 180 ry 0 rz 0.01 deg; joints [38.431, -42.274, 99.435, -136.876, 65.443, 159.62]
  MoveL 5536 to (-170.68, 268.42, -44.5) mm, rotated rx -180 ry 0 rz 0.01 deg; joints [38.449, -42.292, 99.472, -136.864, 65.464, 159.628]
  MoveL 5537 to (-167.48, 269.46, -44.5) mm, rotated rx 180 ry 0 rz 0.01 deg; joints [38.553, -42.376, 99.652, -136.788, 65.572, 159.654]
  MoveL 5538 to (-167.08, 269.62, -44.5) mm, rotated rx 180 ry 0 rz 0.01 deg; joints [38.567, -42.386, 99.673, -136.777, 65.585, 159.656]
  MoveL 5539 to (-163.39, 271.36, -44.5) mm, rotated rx -180 ry 0 rz 0.01 deg; joints [38.703, -42.468, 99.846, -136.667, 65.702, 159.666]
  MoveL 5540 to (-162.81, 271.71, -44.5) mm, rotated rx -180 ry 0 rz 0.01 deg; joints [38.727, -42.479, 99.869, -136.646, 65.719, 159.665]
  MoveL 5541 to (-157, 276.04, -44.5) mm, rotated rx 180 ry 0 rz 0.01 deg; joints [38.988, -42.564, 100.043, -136.408, 65.881, 159.621]
  MoveL 5542 to (-156.44, 276.57, -44.5) mm, rotated rx 180 ry 0 rz 0.01 deg; joints [39.016, -42.569, 100.053, -136.381, 65.895, 159.613]
  MoveL 5543 to (-152.87, 280.78, -44.5) mm, rotated rx -180 ry 0 rz 0.01 deg; joints [39.222, -42.577, 100.064, -136.173, 65.973, 159.527]
  MoveL 5544 to (-152.5, 281.31, -44.5) mm, rotated rx -180 ry 0 rz 0.01 deg; joints [39.246, -42.575, 100.06, -136.147, 65.98, 159.515]
  MoveL 5545 to (-149.77, 286.17, -44.5) mm, rotated rx -180 ry 0 rz 0.01 deg; joints [39.45, -42.535, 99.966, -135.924, 66.018, 159.388]
  MoveL 5546 to (-149.43, 287.04, -44.5) mm, rotated rx 180 ry 0 rz 0.01 deg; joints [39.483, -42.523, 99.938, -135.885, 66.019, 159.362]
  MoveL 5547 to (-147.12, 296.84, -44.5) mm, rotated rx -180 ry 0 rz 0.01 deg; joints [39.818, -42.329, 99.508, -135.472, 65.977, 159.039]
  MoveL 5548 to (-147.03, 297.46, -44.5) mm, rotated rx 180 ry 0 rz 0.01 deg; joints [39.838, -42.315, 99.476, -135.447, 65.972, 159.018]
  MoveL 5549 to (-146.99, 298.18, -44.5) mm, rotated rx -180 ry 0 rz 0.01 deg; joints [39.859, -42.295, 99.434, -135.418, 65.963, 158.991]
  MoveL 5550 to (-147.03, 298.84, -44.5) mm, rotated rx 180 ry 0 rz 0.01 deg; joints [39.877, -42.276, 99.391, -135.392, 65.954, 158.965]
  MoveL 5551 to (-148.48, 308.63, -44.5) mm, rotated rx 180 ry 0 rz 0.01 deg; joints [40.12, -41.947, 98.673, -135.024, 65.77, 158.561]
  MoveL 5552 to (-148.63, 309.24, -44.5) mm, rotated rx 180 ry 0 rz 0.01 deg; joints [40.134, -41.925, 98.623, -135.001, 65.757, 158.535]
  MoveL 5553 to (-149.26, 311.05, -44.5) mm, rotated rx 180 ry 0 rz 0.01 deg; joints [40.17, -41.851, 98.463, -134.937, 65.71, 158.452]
  MoveL 5554 to (-149.45, 311.51, -44.5) mm, rotated rx -180 ry 0 rz 0.01 deg; joints [40.178, -41.831, 98.419, -134.921, 65.696, 158.43]
  MoveL 5555 to (-151.34, 315.14, -44.5) mm, rotated rx 180 ry 0 rz 0.01 deg; joints [40.235, -41.66, 98.05, -134.8, 65.578, 158.251]
  MoveL 5556 to (-151.4, 315.25, -44.5) mm, rotated rx -180 ry 0 rz 0.01 deg; joints [40.237, -41.655, 98.038, -134.796, 65.574, 158.245]
  MoveL 5557 to (-155.13, 321.78, -44.5) mm, rotated rx 180 ry 0 rz 0.01 deg; joints [40.331, -41.334, 97.344, -134.58, 65.349, 157.913]
  MoveL 5558 to (-155.39, 322.17, -44.5) mm, rotated rx 180 ry 0 rz 0.01 deg; joints [40.336, -41.314, 97.3, -134.567, 65.334, 157.892]
  MoveL 5559 to (-156.51, 323.62, -44.5) mm, rotated rx 180 ry 0 rz 0.01 deg; joints [40.35, -41.232, 97.123, -134.522, 65.273, 157.812]
  MoveL 5560 to (-156.86, 324.01, -44.5) mm, rotated rx 180 ry 0 rz 0.01 deg; joints [40.352, -41.208, 97.071, -134.51, 65.255, 157.789]
  MoveL 5561 to (-165.05, 331.75, -44.5) mm, rotated rx 180 ry 0 rz 0.01 deg; joints [40.374, -40.69, 95.955, -134.29, 64.845, 157.309]
  MoveL 5562 to (-165.39, 332.03, -44.5) mm, rotated rx 180 ry 0 rz 0.01 deg; joints [40.373, -40.669, 95.911, -134.282, 64.829, 157.29]
  MoveL 5563 to (-166.84, 333.08, -44.5) mm, rotated rx 180 ry 0 rz 0.01 deg; joints [40.368, -40.586, 95.733, -134.255, 64.76, 157.217]
  MoveL 5564 to (-167.34, 333.38, -44.5) mm, rotated rx 180 ry 0 rz 0.01 deg; joints [40.365, -40.559, 95.675, -134.248, 64.737, 157.194]
  MoveL 5565 to (-177.86, 338.5, -44.5) mm, rotated rx 180 ry 0 rz 0.01 deg; joints [40.26, -40.026, 94.535, -134.146, 64.27, 156.758]
  MoveL 5566 to (-178.27, 338.66, -44.5) mm, rotated rx 180 ry 0 rz 0.01 deg; joints [40.255, -40.006, 94.492, -134.143, 64.253, 156.742]
  MoveL 5567 to (-179.36, 339.03, -44.5) mm, rotated rx 180 ry 0 rz 0.01 deg; joints [40.24, -39.956, 94.384, -134.139, 64.206, 156.703]
  MoveL 5568 to (-179.92, 339.17, -44.5) mm, rotated rx 180 ry 0 rz 0.01 deg; joints [40.231, -39.931, 94.331, -134.138, 64.183, 156.685]
  MoveL 5569 to (-180.17, 339.2, -44.5) mm, rotated rx -180 ry 0 rz 0.01 deg; joints [40.226, -39.921, 94.31, -134.139, 64.173, 156.678]
  MoveL 5570 to (4.87, 339.21, -44.5) mm, rotated rx 180 ry 0 rz 0.01 deg; joints [44.918, -45.994, 107.349, -131.573, 70.74, 160.363]
  MoveL 5571 to (5.94, 339.15, -44.5) mm, rotated rx -180 ry 0 rz 0.01 deg; joints [44.946, -46.027, 107.421, -131.556, 70.776, 160.384]
  MoveL 5572 to (6.8, 338.95, -44.5) mm, rotated rx 180 ry 0 rz 0.01 deg; joints [44.964, -46.058, 107.489, -131.547, 70.807, 160.407]
  MoveL 5573 to (7.07, 338.84, -44.5) mm, rotated rx -180 ry 0 rz 0.01 deg; joints [44.969, -46.069, 107.513, -131.546, 70.817, 160.416]
  MoveL 5574 to (7.57, 338.46, -44.33) mm, rotated rx -180 ry 0 rz 0.01 deg; joints [44.972, -46.104, 107.571, -131.549, 70.833, 160.433]
  MoveL 5575 to (7.78, 338.05, -43.87) mm, rotated rx 180 ry 0 rz 0.01 deg; joints [44.966, -46.147, 107.613, -131.554, 70.83, 160.434]
  MoveL 5576 to (7.82, 337.88, -43.23) mm, rotated rx -180 ry 0 rz 0.01 deg; joints [44.962, -46.188, 107.629, -131.552, 70.813, 160.417]
  Set speed (500.0 mm/s)
  MoveL 5577 to (7.82, 337.88, 11) mm, rotated rx 180 ry 0 rz 0.01 deg; joints [44.942, -49.073, 107.797, -130.824, 69.015, 158.246]
  Set speed (500.0 mm/s)
  MoveL 5578 to (10.27, 334.35, 11) mm, rotated rx -180 ry 0 rz 0.01 deg; joints [44.912, -49.257, 108.178, -130.911, 69.133, 158.417]
  Set speed (100.0 mm/s)
  MoveL 5579 to (10.27, 334.35, -29) mm, rotated rx 180 ry 0 rz 0.01 deg; joints [44.927, -47.131, 108.078, -131.457, 70.473, 160.036]
  MoveL 5580 to (10.27, 334.35, -44.5) mm, rotated rx 180 ry 0 rz 0.01 deg; joints [44.932, -46.291, 108.004, -131.652, 70.982, 160.641]
  MoveL 5581 to (10.27, 31.93, -44.5) mm, rotated rx -180 ry 0 rz 0.01 deg; joints [35.138, -53.453, 124.59, -143.468, 75.28, 170.283]
  MoveL 5582 to (9.28, 36.11, -44.5) mm, rotated rx -180 ry 0 rz 0.01 deg; joints [35.268, -53.345, 124.33, -143.313, 75.183, 170.155]
  MoveL 5583 to (9.16, 36.53, -44.5) mm, rotated rx 180 ry 0 rz 0.01 deg; joints [35.28, -53.334, 124.302, -143.298, 75.172, 170.141]
  MoveL 5584 to (8.5, 38.25, -44.5) mm, rotated rx -180 ry 0 rz 0.01 deg; joints [35.326, -53.282, 124.178, -143.24, 75.124, 170.084]
  MoveL 5585 to (8.27, 38.74, -44.5) mm, rotated rx -180 ry 0 rz 0.01 deg; joints [35.338, -53.266, 124.14, -143.224, 75.108, 170.067]
  MoveL 5586 to (6.11, 42.48, -44.5) mm, rotated rx -180 ry 0 rz 0.01 deg; joints [35.42, -53.132, 123.822, -143.112, 74.977, 169.931]
  MoveL 5587 to (6.08, 42.53, -44.5) mm, rotated rx -180 ry 0 rz 0.01 deg; joints [35.421, -53.13, 123.818, -143.11, 74.976, 169.929]
  MoveL 5588 to (2.59, 48.34, -44.5) mm, rotated rx -180 ry 0 rz 0.01 deg; joints [35.543, -52.916, 123.313, -142.939, 74.767, 169.714]
  MoveL 5589 to (2.35, 48.68, -44.5) mm, rotated rx 180 ry 0 rz 0.01 deg; joints [35.549, -52.903, 123.282, -142.93, 74.754, 169.701]
  MoveL 5590 to (1.03, 50.37, -44.5) mm, rotated rx -180 ry 0 rz 0.01 deg; joints [35.576, -52.832, 123.114, -142.887, 74.683, 169.633]
  MoveL 5591 to (0.48, 50.92, -44.5) mm, rotated rx -180 ry 0 rz 0.01 deg; joints [35.582, -52.805, 123.052, -142.875, 74.656, 169.609]
  MoveL 5592 to (-7.44, 57.29, -44.5) mm, rotated rx -180 ry 0 rz 0.01 deg; joints [35.608, -52.45, 122.223, -142.769, 74.284, 169.305]
  MoveL 5593 to (-7.81, 57.55, -44.5) mm, rotated rx 180 ry 0 rz 0.01 deg; joints [35.607, -52.434, 122.186, -142.766, 74.267, 169.292]
  MoveL 5594 to (-8.47, 57.96, -44.5) mm, rotated rx 180 ry 0 rz 0.01 deg; joints [35.605, -52.406, 122.123, -142.762, 74.238, 169.27]
  MoveL 5595 to (-9.24, 58.3, -44.5) mm, rotated rx -180 ry 0 rz 0.01 deg; joints [35.597, -52.377, 122.055, -142.764, 74.206, 169.248]
  MoveL 5596 to (-19.1, 61.28, -44.5) mm, rotated rx -180 ry 0 rz 0.01 deg; joints [35.451, -52.028, 121.254, -142.834, 73.814, 169.006]
  MoveL 5597 to (-20.03, 61.42, -44.5) mm, rotated rx 180 ry 0 rz 0.01 deg; joints [35.432, -51.998, 121.184, -142.846, 73.779, 168.987]
  MoveL 5598 to (-25.47, 61.49, -44.5) mm, rotated rx 180 ry 0 rz 0.01 deg; joints [35.296, -51.835, 120.814, -142.947, 73.584, 168.897]
  MoveL 5599 to (-26.11, 61.44, -44.5) mm, rotated rx -180 ry 0 rz 0.01 deg; joints [35.278, -51.817, 120.774, -142.962, 73.562, 168.888]
  MoveL 5600 to (-31.56, 60.47, -44.5) mm, rotated rx 180 ry 0 rz 0.01 deg; joints [35.106, -51.675, 120.452, -143.105, 73.382, 168.828]
  MoveL 5601 to (-32.28, 60.26, -44.5) mm, rotated rx -180 ry 0 rz 0.01 deg; joints [35.08, -51.657, 120.413, -143.128, 73.359, 168.822]
  MoveL 5602 to (-38.81, 57.48, -44.5) mm, rotated rx 180 ry 0 rz 0.01 deg; joints [34.817, -51.517, 120.101, -143.365, 73.164, 168.795]
  MoveL 5603 to (-39.36, 57.19, -44.5) mm, rotated rx 180 ry 0 rz 0.01 deg; joints [34.793, -51.506, 120.077, -143.387, 73.149, 168.794]
  MoveL 5604 to (-42.33, 55.21, -44.5) mm, rotated rx -180 ry 0 rz 0.01 deg; joints [34.649, -51.456, 119.968, -143.524, 73.07, 168.802]
  MoveL 5605 to (-42.68, 54.95, -44.5) mm, rotated rx -180 ry 0 rz 0.01 deg; joints [34.631, -51.451, 119.957, -143.541, 73.061, 168.803]
  MoveL 5606 to (-45.69, 52.33, -44.5) mm, rotated rx 180 ry 0 rz 0.01 deg; joints [34.462, -51.412, 119.874, -143.705, 72.989, 168.828]
  MoveL 5607 to (-46.15, 51.84, -44.5) mm, rotated rx 180 ry 0 rz 0.01 deg; joints [34.433, -51.407, 119.865, -143.734, 72.979, 168.835]
  MoveL 5608 to (-50.4, 46.32, -44.5) mm, rotated rx 180 ry 0 rz 0.01 deg; joints [34.131, -51.387, 119.832, -144.04, 72.903, 168.92]
  MoveL 5609 to (-50.64, 45.95, -44.5) mm, rotated rx -180 ry 0 rz 0.01 deg; joints [34.111, -51.387, 119.832, -144.06, 72.899, 168.927]
  MoveL 5610 to (-68.79, 14.55, -44.5) mm, rotated rx 180 ry 0 rz 0.01 deg; joints [32.535, -51.43, 120.002, -145.696, 72.671, 169.498]
  MoveL 5611 to (-68.98, 14.16, -44.5) mm, rotated rx 180 ry 0 rz 0.01 deg; joints [32.516, -51.431, 120.006, -145.716, 72.669, 169.505]
  MoveL 5612 to (-71.72, 7.62, -44.5) mm, rotated rx -180 ry 0 rz 0.01 deg; joints [32.211, -51.468, 120.104, -146.039, 72.657, 169.638]
  MoveL 5613 to (-71.91, 7.02, -44.5) mm, rotated rx 180 ry 0 rz 0.01 deg; joints [32.184, -51.473, 120.117, -146.068, 72.659, 169.651]
  MoveL 5614 to (-72.6, 3.77, -44.5) mm, rotated rx 180 ry 0 rz 0.01 deg; joints [32.048, -51.512, 120.212, -146.218, 72.678, 169.727]
  MoveL 5615 to (-72.66, 3.36, -44.5) mm, rotated rx -180 ry 0 rz 0.01 deg; joints [32.032, -51.517, 120.225, -146.236, 72.681, 169.736]
  MoveL 5616 to (-73.01, -0.63, -44.5) mm, rotated rx 180 ry 0 rz 0.01 deg; joints [31.876, -51.579, 120.375, -146.411, 72.723, 169.837]
  MoveL 5617 to (-73.01, -1.31, -44.5) mm, rotated rx 180 ry 0 rz 0.01 deg; joints [31.85, -51.592, 120.406, -146.44, 72.733, 169.855]
  MoveL 5618 to (-72.17, -8.57, -44.5) mm, rotated rx -180 ry 0 rz 0.01 deg; joints [31.599, -51.749, 120.779, -146.735, 72.864, 170.059]
  MoveL 5619 to (-72, -9.3, -44.5) mm, rotated rx -180 ry 0 rz 0.01 deg; joints [31.576, -51.767, 120.823, -146.763, 72.88, 170.081]
  MoveL 5620 to (-70.78, -12.78, -44.5) mm, rotated rx 180 ry 0 rz 0.01 deg; joints [31.473, -51.867, 121.058, -146.891, 72.974, 170.19]
  MoveL 5621 to (-70.16, -14.48, -44.5) mm, rotated rx 180 ry 0 rz 0.01 deg; joints [31.424, -51.916, 121.175, -146.953, 73.02, 170.244]
  MoveL 5622 to (-69.92, -15.02, -44.5) mm, rotated rx 180 ry 0 rz 0.01 deg; joints [31.409, -51.933, 121.215, -146.972, 73.037, 170.262]
  MoveL 5623 to (-67.66, -18.94, -44.5) mm, rotated rx 180 ry 0 rz 0.01 deg; joints [31.313, -52.072, 121.542, -147.101, 73.176, 170.398]
  MoveL 5624 to (-67.54, -19.13, -44.5) mm, rotated rx 180 ry 0 rz 0.01 deg; joints [31.309, -52.08, 121.558, -147.107, 73.183, 170.405]
  MoveL 5625 to (-66.79, -20.25, -44.5) mm, rotated rx 180 ry 0 rz 0.01 deg; joints [31.284, -52.122, 121.658, -147.142, 73.227, 170.445]
  MoveL 5626 to (-66.3, -20.83, -44.5) mm, rotated rx -180 ry 0 rz 0.01 deg; joints [31.273, -52.148, 121.718, -147.159, 73.253, 170.468]
  MoveL 5627 to (-59.76, -26.98, -44.5) mm, rotated rx -180 ry 0 rz 0.01 deg; joints [31.19, -52.455, 122.436, -147.31, 73.583, 170.725]
  MoveL 5628 to (-59.6, -27.12, -44.5) mm, rotated rx 180 ry 0 rz 0.01 deg; joints [31.188, -52.463, 122.454, -147.314, 73.591, 170.731]
  MoveL 5629 to (-58.51, -28.02, -44.5) mm, rotated rx -180 ry 0 rz 0.01 deg; joints [31.179, -52.512, 122.568, -147.333, 73.644, 170.77]
  MoveC 5630 to (-58.08, -28.32, -44.5) mm, rotated rx 180 ry 0 rz 0.01 deg; joints [31.177, -52.53, 122.611, -147.339, 73.665, 170.785] to (-57.61, -28.56, -44.5) mm, rotated rx -180 ry 0 rz 0.01 deg; joints [31.179, -52.548, 122.654, -147.341, 73.686, 170.798]
  MoveL 5631 to (-50.81, -31.27, -44.5) mm, rotated rx 180 ry 0 rz 0.01 deg; joints [31.234, -52.802, 123.242, -147.338, 73.978, 170.97]
  MoveL 5632 to (-342.73, -31.27, -44.5) mm, rotated rx 180 ry 0 rz 0.01 deg; joints [25.564, -42.612, 100.698, -150.763, 62.119, 166.416]
  MoveL 5633 to (-336.29, -28.75, -44.5) mm, rotated rx 180 ry 0 rz 0.01 deg; joints [25.753, -42.824, 101.148, -150.618, 62.376, 166.45]
  MoveL 5634 to (-335.79, -28.51, -44.5) mm, rotated rx 180 ry 0 rz 0.01 deg; joints [25.77, -42.84, 101.181, -150.604, 62.396, 166.451]
  MoveL 5635 to (-335.06, -28.08, -44.5) mm, rotated rx -180 ry 0 rz 0.01 deg; joints [25.796, -42.861, 101.226, -150.582, 62.423, 166.45]
  MoveL 5636 to (-334.48, -27.64, -44.5) mm, rotated rx 180 ry 0 rz 0.01 deg; joints [25.82, -42.876, 101.257, -150.56, 62.444, 166.447]
  MoveL 5637 to (-327.58, -21.19, -44.5) mm, rotated rx -180 ry 0 rz 0.01 deg; joints [26.152, -43.031, 101.58, -150.242, 62.674, 166.37]
  MoveL 5638 to (-327.34, -20.95, -44.5) mm, rotated rx -180 ry 0 rz 0.01 deg; joints [26.164, -43.036, 101.589, -150.23, 62.682, 166.366]
  MoveL 5639 to (-326.72, -20.24, -44.5) mm, rotated rx -180 ry 0 rz 0.01 deg; joints [26.198, -43.047, 101.613, -150.195, 62.701, 166.355]
  MoveL 5640 to (-326.35, -19.73, -44.5) mm, rotated rx 180 ry 0 rz 0.01 deg; joints [26.222, -43.053, 101.623, -150.171, 62.711, 166.346]
  MoveL 5641 to (-323.78, -15.39, -44.5) mm, rotated rx 180 ry 0 rz 0.01 deg; joints [26.411, -43.074, 101.66, -149.97, 62.774, 166.259]
  MoveL 5642 to (-323.51, -14.82, -44.5) mm, rotated rx -180 ry 0 rz 0.01 deg; joints [26.435, -43.074, 101.659, -149.944, 62.779, 166.246]
  MoveL 5643 to (-321.52, -9.33, -44.5) mm, rotated rx -180 ry 0 rz 0.01 deg; joints [26.653, -43.049, 101.595, -149.697, 62.803, 166.114]
  MoveL 5644 to (-321.34, -8.58, -44.5) mm, rotated rx -180 ry 0 rz 0.01 deg; joints [26.681, -43.042, 101.578, -149.664, 62.802, 166.094]
  MoveL 5645 to (-320.52, -1.69, -44.5) mm, rotated rx 180 ry 0 rz 0.01 deg; joints [26.926, -42.944, 101.353, -149.365, 62.758, 165.897]
  MoveL 5646 to (-320.5, -1.07, -44.5) mm, rotated rx 180 ry 0 rz 0.01 deg; joints [26.947, -42.933, 101.328, -149.338, 62.751, 165.879]
  MoveL 5647 to (-320.74, 2.55, -44.5) mm, rotated rx -180 ry 0 rz 0.01 deg; joints [27.064, -42.854, 101.152, -149.186, 62.699, 165.763]
  MoveL 5648 to (-320.8, 3, -44.5) mm, rotated rx -180 ry 0 rz 0.01 deg; joints [27.078, -42.843, 101.127, -149.167, 62.691, 165.748]
  MoveL 5649 to (-321.6, 6.98, -44.5) mm, rotated rx 180 ry 0 rz 0.01 deg; joints [27.197, -42.735, 100.887, -149.003, 62.61, 165.611]
  MoveL 5650 to (-321.79, 7.61, -44.5) mm, rotated rx 180 ry 0 rz 0.01 deg; joints [27.215, -42.715, 100.843, -148.977, 62.594, 165.588]
  MoveL 5651 to (-324.35, 13.79, -44.5) mm, rotated rx -180 ry 0 rz 0.01 deg; joints [27.376, -42.494, 100.355, -148.73, 62.41, 165.35]
  MoveL 5652 to (-324.54, 14.18, -44.5) mm, rotated rx 180 ry 0 rz 0.01 deg; joints [27.386, -42.478, 100.321, -148.715, 62.397, 165.334]
  MoveL 5653 to (-342.68, 45.66, -44.5) mm, rotated rx -180 ry 0 rz 0.01 deg; joints [28.103, -41.114, 97.338, -147.477, 61.228, 163.988]
  MoveL 5654 to (-342.92, 46.01, -44.5) mm, rotated rx 180 ry 0 rz 0.01 deg; joints [28.11, -41.097, 97.301, -147.464, 61.214, 163.972]
  MoveL 5655 to (-347.09, 51.54, -44.5) mm, rotated rx -180 ry 0 rz 0.01 deg; joints [28.216, -40.811, 96.68, -147.249, 60.964, 163.708]
  MoveL 5656 to (-347.51, 51.99, -44.5) mm, rotated rx 180 ry 0 rz 0.01 deg; joints [28.223, -40.784, 96.622, -147.231, 60.94, 163.685]
  MoveL 5657 to (-350.26, 54.51, -44.5) mm, rotated rx -180 ry 0 rz 0.01 deg; joints [28.257, -40.618, 96.263, -147.137, 60.788, 163.547]
  MoveL 5658 to (-350.61, 54.79, -44.5) mm, rotated rx -180 ry 0 rz 0.01 deg; joints [28.26, -40.598, 96.219, -147.126, 60.769, 163.531]
  MoveL 5659 to (-353.73, 56.95, -44.5) mm, rotated rx -180 ry 0 rz 0.01 deg; joints [28.275, -40.423, 95.843, -147.048, 60.604, 163.397]
  MoveL 5660 to (-354.3, 57.27, -44.5) mm, rotated rx -180 ry 0 rz 0.01 deg; joints [28.276, -40.393, 95.778, -147.037, 60.575, 163.375]
  MoveL 5661 to (-360.83, 60.14, -44.5) mm, rotated rx 180 ry 0 rz 0.01 deg; joints [28.255, -40.061, 95.065, -146.941, 60.25, 163.148]
  MoveL 5662 to (-361.57, 60.37, -44.5) mm, rotated rx -180 ry 0 rz 0.01 deg; joints [28.25, -40.025, 94.988, -146.934, 60.213, 163.125]
  MoveL 5663 to (-367.38, 61.44, -44.5) mm, rotated rx 180 ry 0 rz 0.01 deg; joints [28.185, -39.759, 94.42, -146.91, 59.94, 162.971]
  MoveL 5664 to (-368.04, 61.49, -44.5) mm, rotated rx 180 ry 0 rz 0.01 deg; joints [28.175, -39.73, 94.359, -146.91, 59.91, 162.956]
  MoveL 5665 to (-373.48, 61.42, -44.5) mm, rotated rx -180 ry 0 rz 0.01 deg; joints [28.081, -39.503, 93.875, -146.932, 59.665, 162.847]
  MoveL 5666 to (-374.4, 61.28, -44.5) mm, rotated rx -180 ry 0 rz 0.01 deg; joints [28.061, -39.467, 93.799, -146.942, 59.625, 162.833]
  MoveL 5667 to (-383.59, 58.54, -44.5) mm, rotated rx -180 ry 0 rz 0.01 deg; joints [27.821, -39.135, 93.099, -147.087, 59.24, 162.737]
  MoveL 5668 to (-383.93, 58.42, -44.5) mm, rotated rx -180 ry 0 rz 0.01 deg; joints [27.812, -39.124, 93.074, -147.093, 59.226, 162.734]
  MoveL 5669 to (-384.92, 58.01, -44.5) mm, rotated rx 180 ry 0 rz 0.01 deg; joints [27.782, -39.09, 93.004, -147.114, 59.185, 162.728]
  MoveL 5670 to (-385.72, 57.54, -44.5) mm, rotated rx 180 ry 0 rz 0.01 deg; joints [27.754, -39.066, 92.954, -147.137, 59.154, 162.727]
  MoveL 5671 to (-393.65, 51.26, -44.5) mm, rotated rx 180 ry 0 rz 0.01 deg; joints [27.426, -38.86, 92.529, -147.428, 58.865, 162.779]
  MoveL 5672 to (-394.13, 50.8, -44.5) mm, rotated rx -180 ry 0 rz 0.01 deg; joints [27.404, -38.85, 92.507, -147.449, 58.848, 162.785]
  MoveL 5673 to (-395.53, 49.15, -44.5) mm, rotated rx 180 ry 0 rz 0.01 deg; joints [27.329, -38.825, 92.456, -147.524, 58.803, 162.813]
  MoveL 5674 to (-395.82, 48.75, -44.5) mm, rotated rx -180 ry 0 rz 0.01 deg; joints [27.312, -38.821, 92.449, -147.542, 58.795, 162.821]
  MoveL 5675 to (-397.86, 45.48, -44.5) mm, rotated rx -180 ry 0 rz 0.01 deg; joints [27.175, -38.802, 92.415, -147.688, 58.739, 162.891]
  MoveL 5676 to (-397.92, 45.39, -44.5) mm, rotated rx -180 ry 0 rz 0.01 deg; joints [27.172, -38.802, 92.415, -147.692, 58.737, 162.893]
  MoveL 5677 to (-401.78, 38.75, -44.5) mm, rotated rx -180 ry 0 rz 0.01 deg; joints [26.9, -38.776, 92.371, -147.988, 58.637, 163.042]
  MoveL 5678 to (-402.01, 38.25, -44.5) mm, rotated rx 180 ry 0 rz 0.01 deg; joints [26.88, -38.776, 92.372, -148.01, 58.631, 163.055]
  MoveL 5679 to (-402.67, 36.53, -44.5) mm, rotated rx 180 ry 0 rz 0.01 deg; joints [26.815, -38.784, 92.392, -148.086, 58.621, 163.1]
  MoveL 5680 to (-402.8, 36.11, -44.5) mm, rotated rx 180 ry 0 rz 0.01 deg; joints [26.8, -38.787, 92.4, -148.105, 58.62, 163.112]
  MoveL 5681 to (-403.78, 31.96, -44.5) mm, rotated rx -180 ry 0 rz 0.01 deg; joints [26.653, -38.831, 92.501, -148.287, 58.623, 163.234]
  MoveL 5682 to (-403.79, 333.8, -44.5) mm, rotated rx -180 ry 0 rz 0.01 deg; joints [35.414, -30.616, 74.785, -134.792, 54.767, 150.779]
  MoveL 5683 to (-403.73, 334.87, -44.5) mm, rotated rx -180 ry 0 rz 0.01 deg; joints [35.444, -30.582, 74.712, -134.742, 54.755, 150.727]
  MoveL 5684 to (-403.53, 335.74, -44.5) mm, rotated rx -180 ry 0 rz 0.01 deg; joints [35.47, -30.561, 74.669, -134.703, 54.752, 150.691]
  MoveL 5685 to (-403.42, 336, -44.5) mm, rotated rx 180 ry 0 rz 0.01 deg; joints [35.479, -30.558, 74.661, -134.691, 54.754, 150.681]
  MoveL 5686 to (-403.03, 336.5, -44.33) mm, rotated rx 180 ry 0 rz 0.01 deg; joints [35.5, -30.567, 74.665, -134.667, 54.761, 150.664]
  MoveL 5687 to (-402.62, 336.71, -43.87) mm, rotated rx -180 ry 0 rz 0.01 deg; joints [35.513, -30.6, 74.695, -134.652, 54.765, 150.653]
  MoveL 5688 to (-402.46, 336.75, -43.23) mm, rotated rx -180 ry 0 rz 0.01 deg; joints [35.517, -30.634, 74.713, -134.639, 54.756, 150.637]
  Set speed (500.0 mm/s)
  MoveL 5689 to (-402.46, 336.75, 11) mm, rotated rx 180 ry 0 rz 0.01 deg; joints [35.493, -32.912, 74.899, -133.574, 53.288, 148.796]
  Set speed (500.0 mm/s)
  MoveL 5690 to (-328.21, 254.07, 11) mm, rotated rx 180 ry 0 rz 0.01 deg; joints [34.659, -39.098, 87.573, -137.593, 57.514, 154.821]
  Set speed (500.0 mm/s)
  MoveL 5691 to (-328.21, 254.07, -32.73) mm, rotated rx -180 ry 0 rz 0.01 deg; joints [34.679, -37.131, 87.452, -138.338, 58.895, 156.265]
  Set speed (100.0 mm/s)
  MoveL 5692 to (-328.05, 254.05, -33.35) mm, rotated rx -180 ry 0 rz 0.01 deg; joints [34.682, -37.11, 87.465, -138.348, 58.922, 156.289]
  MoveL 5693 to (-327.6, 254.02, -33.82) mm, rotated rx 180 ry 0 rz 0.01 deg; joints [34.69, -37.108, 87.504, -138.356, 58.956, 156.316]
  MoveL 5694 to (-326.99, 254.04, -34) mm, rotated rx -180 ry 0 rz 0.01 deg; joints [34.703, -37.126, 87.558, -138.357, 58.988, 156.337]
  MoveL 5695 to (-321.75, 258.06, -34.24) mm, rotated rx -180 ry 0 rz 0.01 deg; joints [34.92, -37.222, 87.774, -138.176, 59.17, 156.311]
  MoveL 5696 to (-323.34, 264.47, -34.49) mm, rotated rx -180 ry 0 rz 0.01 deg; joints [35.07, -36.956, 87.232, -137.907, 59.028, 156.012]
  MoveL 5697 to (-329.85, 265.59, -34.73) mm, rotated rx 180 ry 0 rz 0.01 deg; joints [34.973, -36.633, 86.577, -137.875, 58.74, 155.806]
  MoveL 5698 to (-333.48, 260.07, -34.98) mm, rotated rx 180 ry 0 rz 0.01 deg; joints [34.747, -36.627, 86.595, -138.124, 58.66, 155.951]
  MoveL 5699 to (-329.87, 254.53, -35.22) mm, rotated rx 180 ry 0 rz 0.01 deg; joints [34.661, -36.932, 87.263, -138.361, 58.894, 156.282]
  MoveL 5700 to (-323.36, 255.61, -35.46) mm, rotated rx 180 ry 0 rz 0.01 deg; joints [34.82, -37.168, 87.777, -138.305, 59.169, 156.41]
  MoveL 5701 to (-321.74, 262.02, -35.71) mm, rotated rx 180 ry 0 rz 0.01 deg; joints [35.033, -37.04, 87.522, -138.029, 59.165, 156.194]
  MoveL 5702 to (-326.96, 266.07, -35.95) mm, rotated rx 180 ry 0 rz 0.01 deg; joints [35.044, -36.688, 86.801, -137.869, 58.896, 155.9]
  MoveL 5703 to (-332.76, 262.91, -36.2) mm, rotated rx -180 ry 0 rz 0.01 deg; joints [34.841, -36.52, 86.476, -138.019, 58.692, 155.89]
  MoveL 5704 to (-332.19, 256.33, -36.44) mm, rotated rx -180 ry 0 rz 0.01 deg; joints [34.667, -36.725, 86.937, -138.307, 58.809, 156.187]
  MoveL 5705 to (-325.93, 254.21, -36.68) mm, rotated rx 180 ry 0 rz 0.01 deg; joints [34.73, -37.042, 87.628, -138.39, 59.114, 156.441]
  MoveL 5706 to (-321.49, 259.1, -36.93) mm, rotated rx -180 ry 0 rz 0.01 deg; joints [34.956, -37.079, 87.72, -138.174, 59.251, 156.36]
  MoveL 5707 to (-324.18, 265.13, -37.17) mm, rotated rx -180 ry 0 rz 0.01 deg; joints [35.073, -36.778, 87.103, -137.924, 59.065, 156.049]
  MoveL 5708 to (-330.78, 265.08, -37.42) mm, rotated rx -180 ry 0 rz 0.01 deg; joints [34.941, -36.485, 86.512, -137.942, 58.788, 155.889]
  MoveL 5709 to (-333.38, 259, -37.66) mm, rotated rx -180 ry 0 rz 0.01 deg; joints [34.72, -36.539, 86.657, -138.213, 58.76, 156.083]
  MoveL 5710 to (-328.86, 254.19, -37.9) mm, rotated rx -180 ry 0 rz 0.01 deg; joints [34.672, -36.862, 87.361, -138.417, 59.025, 156.407]
  MoveL 5711 to (-322.64, 256.4, -38.15) mm, rotated rx 180 ry 0 rz 0.01 deg; joints [34.857, -37.052, 87.779, -138.311, 59.273, 156.48]
  MoveL 5712 to (-322.17, 262.99, -38.39) mm, rotated rx 180 ry 0 rz 0.01 deg; joints [35.053, -36.87, 87.409, -138.031, 59.217, 156.228]
  MoveL 5713 to (-328.02, 266.06, -38.64) mm, rotated rx 180 ry 0 rz 0.01 deg; joints [35.024, -36.519, 86.693, -137.914, 58.932, 155.958]
  MoveL 5714 to (-333.18, 261.93, -38.88) mm, rotated rx 180 ry 0 rz 0.01 deg; joints [34.807, -36.407, 86.486, -138.106, 58.769, 156.005]
  MoveL 5715 to (-331.46, 255.55, -39.13) mm, rotated rx -180 ry 0 rz 0.01 deg; joints [34.66, -36.655, 87.038, -138.382, 58.933, 156.323]
  MoveL 5716 to (-324.93, 254.57, -39.37) mm, rotated rx -180 ry 0 rz 0.01 deg; joints [34.761, -36.951, 87.682, -138.415, 59.236, 156.537]
  MoveL 5717 to (-321.41, 260.16, -39.61) mm, rotated rx 180 ry 0 rz 0.01 deg; joints [34.989, -36.928, 87.648, -138.17, 59.323, 156.403]
  MoveL 5718 to (-325.12, 265.62, -39.86) mm, rotated rx 180 ry 0 rz 0.01 deg; joints [35.069, -36.6, 86.974, -137.947, 59.1, 156.089]
  MoveL 5719 to (-331.62, 264.41, -40.1) mm, rotated rx 180 ry 0 rz 0.01 deg; joints [34.908, -36.346, 86.465, -138.015, 58.842, 155.98]
  MoveL 5720 to (-333.11, 257.97, -40.35) mm, rotated rx 180 ry 0 rz 0.01 deg; joints [34.697, -36.458, 86.732, -138.3, 58.867, 156.218]
  MoveL 5721 to (-327.81, 254.03, -40.59) mm, rotated rx -180 ry 0 rz 0.01 deg; joints [34.69, -36.787, 87.452, -138.464, 59.156, 156.524]
  MoveL 5722 to (-322.07, 257.3, -40.83) mm, rotated rx -180 ry 0 rz 0.01 deg; joints [34.895, -36.926, 87.76, -138.313, 59.369, 156.542]
  MoveL 5723 to (-322.77, 263.87, -41.08) mm, rotated rx 180 ry 0 rz 0.01 deg; joints [35.067, -36.695, 87.287, -138.037, 59.262, 156.26]
  MoveL 5724 to (-329.07, 265.86, -41.32) mm, rotated rx 180 ry 0 rz 0.01 deg; joints [34.999, -36.357, 86.597, -137.968, 58.971, 156.023]
  MoveL 5725 to (-333.42, 260.89, -41.57) mm, rotated rx 180 ry 0 rz 0.01 deg; joints [34.774, -36.304, 86.516, -138.194, 58.853, 156.126]
  MoveL 5726 to (-330.6, 254.91, -41.81) mm, rotated rx 180 ry 0 rz 0.01 deg; joints [34.66, -36.587, 87.14, -138.45, 59.061, 156.455]
  MoveL 5727 to (-324, 255.1, -42.05) mm, rotated rx -180 ry 0 rz 0.01 deg; joints [34.795, -36.851, 87.718, -138.432, 59.352, 156.623]
  MoveL 5728 to (-321.53, 261.22, -42.3) mm, rotated rx -180 ry 0 rz 0.01 deg; joints [35.018, -36.768, 87.557, -138.167, 59.387, 156.441]
  MoveL 5729 to (-326.14, 265.94, -42.54) mm, rotated rx 180 ry 0 rz 0.01 deg; joints [35.06, -36.424, 86.848, -137.978, 59.134, 156.134]
  MoveL 5730 to (-332.32, 263.61, -42.79) mm, rotated rx 180 ry 0 rz 0.01 deg; joints [34.872, -36.216, 86.438, -138.094, 58.903, 156.08]
  MoveL 5731 to (-332.65, 257.01, -43.03) mm, rotated rx 180 ry 0 rz 0.01 deg; joints [34.68, -36.382, 86.819, -138.383, 58.982, 156.354]
  MoveL 5732 to (-326.74, 254.06, -43.27) mm, rotated rx 180 ry 0 rz 0.01 deg; joints [34.713, -36.708, 87.531, -138.502, 59.284, 156.634]
  MoveL 5733 to (-321.67, 258.29, -43.52) mm, rotated rx 180 ry 0 rz 0.01 deg; joints [34.932, -36.79, 87.72, -138.312, 59.456, 156.596]
  MoveL 5734 to (-323.52, 264.63, -43.76) mm, rotated rx 180 ry 0 rz 0.01 deg; joints [35.075, -36.517, 87.158, -138.048, 59.301, 156.294]
  MoveL 5735 to (-330.07, 265.48, -44.01) mm, rotated rx 180 ry 0 rz 0.01 deg; joints [34.97, -36.202, 86.516, -138.028, 59.014, 156.098]
  MoveL 5736 to (-333.47, 259.82, -44.25) mm, rotated rx 180 ry 0 rz 0.01 deg; joints [34.744, -36.209, 86.563, -138.282, 58.947, 156.253]
  MoveL 5737 to (-329.65, 254.44, -44.49) mm, rotated rx -180 ry 0 rz 0.01 deg; joints [34.667, -36.517, 87.241, -138.511, 59.191, 156.583]
  MoveL 5738 to (-323.18, 255.78, -44.74) mm, rotated rx 180 ry 0 rz 0.01 deg; joints [34.832, -36.742, 87.734, -138.442, 59.461, 156.699]
  MoveL 5739 to (-321.82, 262.24, -44.98) mm, rotated rx 180 ry 0 rz 0.01 deg; joints [35.042, -36.602, 87.452, -138.166, 59.443, 156.475]
  MoveL 5740 to (-327.2, 266.08, -45.23) mm, rotated rx 180 ry 0 rz 0.01 deg; joints [35.044, -36.251, 86.73, -138.016, 59.168, 156.185]
  MoveL 5741 to (-332.87, 262.69, -45.47) mm, rotated rx 180 ry 0 rz 0.01 deg; joints [34.837, -36.096, 86.431, -138.176, 58.973, 156.187]
  MoveL 5742 to (-332.04, 256.14, -45.71) mm, rotated rx 180 ry 0 rz 0.01 deg; joints [34.669, -36.31, 86.914, -138.462, 59.102, 156.489]
  MoveL 5743 to (-325.7, 254.28, -45.96) mm, rotated rx -180 ry 0 rz 0.01 deg; joints [34.741, -36.622, 87.596, -138.532, 59.409, 156.735]
  MoveL 5744 to (-321.45, 259.34, -46.2) mm, rotated rx 180 ry 0 rz 0.01 deg; joints [34.968, -36.645, 87.659, -138.308, 59.534, 156.642]
  MoveL 5745 to (-324.39, 265.25, -46.45) mm, rotated rx 180 ry 0 rz 0.01 deg; joints [35.077, -36.338, 87.027, -138.065, 59.337, 156.33]
  MoveL 5746 to (-330.98, 264.94, -46.69) mm, rotated rx 180 ry 0 rz 0.01 deg; joints [34.938, -36.055, 86.453, -138.095, 59.062, 156.181]
  MoveL 5747 to (-333.34, 258.77, -46.93) mm, rotated rx 180 ry 0 rz 0.01 deg; joints [34.718, -36.122, 86.626, -138.37, 59.048, 156.384]
  MoveL 5748 to (-328.63, 254.14, -47.18) mm, rotated rx 180 ry 0 rz 0.01 deg; joints [34.68, -36.445, 87.336, -138.563, 59.322, 156.705]
  MoveL 5749 to (-322.5, 256.6, -47.42) mm, rotated rx -180 ry 0 rz 0.01 deg; joints [34.87, -36.622, 87.729, -138.447, 59.563, 156.766]
  MoveL 5750 to (-322.3, 263.2, -47.67) mm, rotated rx 180 ry 0 rz 0.01 deg; joints [35.061, -36.43, 87.335, -138.167, 59.492, 156.507]
  MoveL 5751 to (-328.27, 266.03, -47.91) mm, rotated rx 180 ry 0 rz 0.01 deg; joints [35.023, -36.083, 86.622, -138.062, 59.203, 156.244]
  MoveL 5752 to (-333.25, 261.69, -48.15) mm, rotated rx -180 ry 0 rz 0.01 deg; joints [34.803, -35.985, 86.444, -138.262, 59.05, 156.303]
  MoveL 5753 to (-331.27, 255.39, -48.4) mm, rotated rx 180 ry 0 rz 0.01 deg; joints [34.664, -36.24, 87.013, -138.534, 59.227, 156.623]
  MoveL 5754 to (-324.71, 254.68, -48.64) mm, rotated rx 180 ry 0 rz 0.01 deg; joints [34.773, -36.527, 87.644, -138.554, 59.53, 156.827]
  MoveL 5755 to (-321.42, 260.4, -48.89) mm, rotated rx 180 ry 0 rz 0.01 deg; joints [35, -36.491, 87.58, -138.304, 59.604, 156.683]
  MoveL 5756 to (-325.35, 265.71, -49.13) mm, rotated rx 180 ry 0 rz 0.01 deg; joints [35.072, -36.16, 86.896, -138.089, 59.371, 156.37]
  MoveL 5757 to (-331.79, 264.24, -49.38) mm, rotated rx -180 ry 0 rz 0.01 deg; joints [34.904, -35.917, 86.409, -138.169, 59.117, 156.272]
  MoveL 5758 to (-333.02, 257.75, -49.62) mm, rotated rx -180 ry 0 rz 0.01 deg; joints [34.697, -36.041, 86.702, -138.455, 59.157, 156.518]
  MoveL 5759 to (-327.57, 254.02, -49.86) mm, rotated rx -180 ry 0 rz 0.01 deg; joints [34.699, -36.369, 87.422, -138.607, 59.451, 156.819]
  MoveL 5760 to (-321.97, 257.52, -50.11) mm, rotated rx -180 ry 0 rz 0.01 deg; joints [34.908, -36.493, 87.703, -138.447, 59.656, 156.825]
  MoveL 5761 to (-322.93, 264.06, -50.35) mm, rotated rx 180 ry 0 rz 0.01 deg; joints [35.073, -36.253, 87.209, -138.173, 59.535, 156.539]
  MoveL 5762 to (-329.31, 265.79, -50.6) mm, rotated rx -180 ry 0 rz 0.01 deg; joints [34.997, -35.921, 86.527, -138.116, 59.242, 156.31]
  MoveL 5763 to (-333.45, 260.65, -50.84) mm, rotated rx 180 ry 0 rz 0.01 deg; joints [34.771, -35.882, 86.475, -138.349, 59.137, 156.424]
  MoveL 5764 to (-330.39, 254.79, -51.08) mm, rotated rx 180 ry 0 rz 0.01 deg; joints [34.665, -36.17, 87.114, -138.599, 59.355, 156.753]
  MoveL 5765 to (-323.8, 255.24, -51.33) mm, rotated rx 180 ry 0 rz 0.01 deg; joints [34.808, -36.424, 87.674, -138.568, 59.644, 156.91]
  MoveL 5766 to (-321.58, 261.46, -51.57) mm, rotated rx 180 ry 0 rz 0.01 deg; joints [35.028, -36.329, 87.485, -138.3, 59.665, 156.718]
  MoveL 5767 to (-326.38, 265.99, -51.82) mm, rotated rx 180 ry 0 rz 0.01 deg; joints [35.06, -35.983, 86.77, -138.121, 59.403, 156.415]
  MoveL 5768 to (-332.46, 263.41, -52.06) mm, rotated rx 180 ry 0 rz 0.01 deg; joints [34.868, -35.788, 86.384, -138.248, 59.18, 156.373]
  MoveL 5769 to (-332.53, 256.8, -52.3) mm, rotated rx 180 ry 0 rz 0.01 deg; joints [34.681, -35.965, 86.789, -138.536, 59.273, 156.653]
  MoveL 5770 to (-326.5, 254.09, -52.55) mm, rotated rx 180 ry 0 rz 0.01 deg; joints [34.723, -36.286, 87.496, -138.643, 59.579, 156.926]
  MoveL 5771 to (-321.61, 258.53, -52.79) mm, rotated rx 180 ry 0 rz 0.01 deg; joints [34.945, -36.355, 87.657, -138.444, 59.74, 156.876]
  MoveL 5772 to (-323.71, 264.79, -53.04) mm, rotated rx -180 ry 0 rz 0.01 deg; joints [35.08, -36.075, 87.077, -138.185, 59.573, 156.572]
  MoveL 5773 to (-330.29, 265.37, -53.28) mm, rotated rx 180 ry 0 rz 0.01 deg; joints [34.967, -35.767, 86.449, -138.178, 59.285, 156.385]
  MoveL 5774 to (-333.46, 259.58, -53.52) mm, rotated rx 180 ry 0 rz 0.01 deg; joints [34.742, -35.788, 86.524, -138.437, 59.232, 156.551]
  MoveL 5775 to (-329.42, 254.35, -53.77) mm, rotated rx 180 ry 0 rz 0.01 deg; joints [34.673, -36.099, 87.211, -138.657, 59.485, 156.878]
  MoveL 5776 to (-323.01, 255.96, -54.01) mm, rotated rx -180 ry 0 rz 0.01 deg; joints [34.845, -36.312, 87.683, -138.576, 59.75, 156.983]
  MoveL 5777 to (-321.92, 262.47, -54.26) mm, rotated rx 180 ry 0 rz 0.01 deg; joints [35.051, -36.16, 87.375, -138.299, 59.718, 156.751]
  MoveL 5778 to (-327.44, 266.08, -54.5) mm, rotated rx 180 ry 0 rz 0.01 deg; joints [35.043, -35.811, 86.652, -138.16, 59.437, 156.467]
  MoveL 5779 to (-327.83, 266.08, -54.5) mm, rotated rx 180 ry 0 rz 0.01 deg; joints [35.036, -35.795, 86.617, -138.161, 59.42, 156.456]
  MoveC 5780 to (-329.84, 265.25, -54.5) mm, rotated rx -180 ry 0 rz 0.01 deg; joints [34.973, -35.733, 86.489, -138.201, 59.343, 156.439] to (-330.67, 263.25, -54.5) mm, rotated rx 180 ry 0 rz 0.01 deg; joints [34.9, -35.756, 86.54, -138.289, 59.334, 156.501]
  MoveL 5781 to (-330.67, 221.14, -54.5) mm, rotated rx 180 ry 0 rz 0.01 deg; joints [33.699, -36.936, 89.106, -140.092, 59.895, 158.208]
  MoveC 5782 to (-329.58, 220, -54.5) mm, rotated rx -180 ry 0 rz 0.01 deg; joints [33.687, -37.012, 89.271, -140.138, 59.957, 158.28] to (-328.38, 221.03, -54.5) mm, rotated rx 180 ry 0 rz 0.01 deg; joints [33.74, -37.034, 89.316, -140.09, 59.996, 158.268]
  MoveL 5783 to (-324.19, 262.96, -54.5) mm, rotated rx -180 ry 0 rz 0.01 deg; joints [35.02, -36.039, 87.139, -138.287, 59.62, 156.68]
  MoveC 5784 to (-324.91, 265.15, -54.5) mm, rotated rx -180 ry 0 rz 0.01 deg; joints [35.067, -35.945, 86.938, -138.195, 59.56, 156.571] to (-327.02, 266.09, -54.5) mm, rotated rx 180 ry 0 rz 0.01 deg; joints [35.052, -35.829, 86.69, -138.159, 59.455, 156.478]
  MoveL 5785 to (-327.44, 266.08, -54.5) mm, rotated rx 180 ry 0 rz 0.01 deg; joints [35.043, -35.811, 86.652, -138.16, 59.437, 156.467]
  MoveC 5786 to (-329.63, 266.88, -54.5) mm, rotated rx -180 ry 0 rz 0.01 deg; joints [35.023, -35.695, 86.405, -138.13, 59.331, 156.377] to (-330.79, 268.89, -54.5) mm, rotated rx 180 ry 0 rz 0.01 deg; joints [35.056, -35.587, 86.173, -138.046, 59.253, 156.262]
  MoveC 5787 to (-332.53, 270.8, -54.5) mm, rotated rx -180 ry 0 rz 0.01 deg; joints [35.076, -35.457, 85.895, -137.966, 59.151, 156.136] to (-335, 270.07, -54.5) mm, rotated rx 180 ry 0 rz 0.01 deg; joints [35.007, -35.372, 85.717, -138.002, 59.052, 156.101]
  MoveC 5788 to (-335.71, 268.88, -54.5) mm, rotated rx 180 ry 0 rz 0.01 deg; joints [34.959, -35.376, 85.728, -138.054, 59.037, 156.132] to (-335.96, 267.52, -54.5) mm, rotated rx -180 ry 0 rz 0.01 deg; joints [34.917, -35.405, 85.791, -138.113, 59.044, 156.183]
  MoveL 5789 to (-335.96, 181.59, -54.5) mm, rotated rx -180 ry 0 rz 0.01 deg; joints [32.439, -37.757, 90.917, -141.796, 60.182, 159.613]
  MoveC 5790 to (-334.85, 179.77, -54.5) mm, rotated rx 180 ry 0 rz 0.01 deg; joints [32.406, -37.85, 91.118, -141.869, 60.254, 159.707] to (-332.72, 179.93, -54.5) mm, rotated rx 180 ry 0 rz 0.01 deg; joints [32.451, -37.934, 91.297, -141.855, 60.345, 159.751]
  MoveL 5791 to (-328.14, 183.22, -54.5) mm, rotated rx 180 ry 0 rz 0.01 deg; joints [32.635, -38.039, 91.516, -141.697, 60.503, 159.732]
  MoveC 5792 to (-327.06, 184.4, -54.5) mm, rotated rx -180 ry 0 rz 0.01 deg; joints [32.691, -38.053, 91.543, -141.642, 60.534, 159.712] to (-326.57, 185.93, -54.5) mm, rotated rx -180 ry 0 rz 0.01 deg; joints [32.746, -38.034, 91.501, -141.576, 60.536, 159.666]
  MoveL 5793 to (-318.41, 267.61, -54.5) mm, rotated rx -180 ry 0 rz 0.01 deg; joints [35.265, -36.148, 87.363, -138.073, 59.809, 156.636]
  MoveC 5794 to (-319.28, 270.25, -54.5) mm, rotated rx 180 ry 0 rz 0.01 deg; joints [35.322, -36.035, 87.12, -137.963, 59.736, 156.504] to (-321.81, 271.38, -54.5) mm, rotated rx -180 ry 0 rz 0.01 deg; joints [35.303, -35.895, 86.823, -137.921, 59.61, 156.392]
  MoveL 5795 to (-332.11, 271.38, -54.5) mm, rotated rx 180 ry 0 rz 0.01 deg; joints [35.1, -35.458, 85.896, -137.941, 59.162, 156.123]
  MoveC 5796 to (-333.7, 271.04, -54.5) mm, rotated rx -180 ry 0 rz 0.01 deg; joints [35.059, -35.4, 85.774, -137.958, 59.097, 156.095] to (-335, 270.07, -54.5) mm, rotated rx 180 ry 0 rz 0.01 deg; joints [35.007, -35.372, 85.717, -138.002, 59.052, 156.101]
  MoveC 5797 to (-337.4, 267.9, -54.5) mm, rotated rx 180 ry 0 rz 0.01 deg; joints [34.899, -35.333, 85.637, -138.099, 58.976, 156.129] to (-340.22, 266.32, -54.5) mm, rotated rx 180 ry 0 rz 0.01 deg; joints [34.8, -35.257, 85.48, -138.171, 58.873, 156.121]
  MoveC 5798 to (-342.8, 264.18, -54.5) mm, rotated rx -180 ry 0 rz 0.01 deg; joints [34.69, -35.208, 85.38, -138.267, 58.788, 156.142] to (-343.77, 260.96, -54.5) mm, rotated rx 180 ry 0 rz 0.01 deg; joints [34.581, -35.26, 85.494, -138.407, 58.788, 156.252]
  MoveL 5799 to (-343.77, 166.36, -54.5) mm, rotated rx 180 ry 0 rz 0.01 deg; joints [31.839, -37.817, 91.071, -142.472, 60.035, 160.006]
  MoveC 5800 to (-342.66, 164.54, -54.5) mm, rotated rx 180 ry 0 rz 0.01 deg; joints [31.805, -37.909, 91.271, -142.546, 60.108, 160.1] to (-340.53, 164.7, -54.5) mm, rotated rx 180 ry 0 rz 0.01 deg; joints [31.85, -37.994, 91.451, -142.531, 60.2, 160.142]
  MoveL 5801 to (-323.78, 176.73, -54.5) mm, rotated rx -180 ry 0 rz 0.01 deg; joints [32.525, -38.382, 92.259, -141.954, 60.777, 160.075]
  MoveC 5802 to (-320.34, 180.52, -54.5) mm, rotated rx -180 ry 0 rz 0.01 deg; joints [32.704, -38.426, 92.347, -141.778, 60.876, 160.011] to (-318.77, 185.39, -54.5) mm, rotated rx -180 ry 0 rz 0.01 deg; joints [32.879, -38.367, 92.211, -141.565, 60.881, 159.864]
  MoveL 5803 to (-309.78, 275.42, -54.5) mm, rotated rx 180 ry 0 rz 0.01 deg; joints [35.657, -36.282, 87.636, -137.716, 60.076, 156.533]
  MoveC 5804 to (-310.65, 278.06, -54.5) mm, rotated rx 180 ry 0 rz 0.01 deg; joints [35.714, -36.169, 87.392, -137.606, 60.003, 156.401] to (-313.18, 279.19, -54.5) mm, rotated rx -180 ry 0 rz 0.01 deg; joints [35.694, -36.03, 87.096, -137.565, 59.878, 156.289]
  MoveL 5805 to (-339.92, 279.19, -54.5) mm, rotated rx -180 ry 0 rz 0.01 deg; joints [35.164, -34.89, 84.685, -137.612, 58.713, 155.582]
  MoveC 5806 to (-342.64, 278.06, -54.5) mm, rotated rx 180 ry 0 rz 0.01 deg; joints [35.08, -34.805, 84.507, -137.663, 58.607, 155.556] to (-343.77, 275.34, -54.5) mm, rotated rx -180 ry 0 rz 0.01 deg; joints [34.982, -34.837, 84.579, -137.783, 58.594, 155.642]
  MoveL 5807 to (-343.77, 260.96, -54.5) mm, rotated rx -180 ry 0 rz 0.01 deg; joints [34.581, -35.26, 85.494, -138.407, 58.788, 156.252]
  MoveC 5808 to (-344.84, 257.44, -54.5) mm, rotated rx 180 ry 0 rz 0.01 deg; joints [34.461, -35.316, 85.617, -138.561, 58.788, 156.371] to (-347.68, 255.11, -54.5) mm, rotated rx 180 ry 0 rz 0.01 deg; joints [34.341, -35.26, 85.503, -138.665, 58.693, 156.394]
  MoveC 5809 to (-350.52, 252.77, -54.5) mm, rotated rx -180 ry 0 rz 0.01 deg; joints [34.22, -35.204, 85.389, -138.769, 58.598, 156.416] to (-351.58, 249.25, -54.5) mm, rotated rx 180 ry 0 rz 0.01 deg; joints [34.1, -35.259, 85.51, -138.923, 58.598, 156.535]
  MoveL 5810 to (-351.58, 151.14, -54.5) mm, rotated rx -180 ry 0 rz 0.01 deg; joints [31.239, -37.869, 91.207, -143.148, 59.885, 160.395]
  MoveC 5811 to (-350.47, 149.32, -54.5) mm, rotated rx 180 ry 0 rz 0.01 deg; joints [31.204, -37.96, 91.404, -143.222, 59.958, 160.487] to (-348.34, 149.48, -54.5) mm, rotated rx -180 ry 0 rz 0.01 deg; joints [31.248, -38.045, 91.586, -143.208, 60.05, 160.53]
  MoveL 5812 to (-316.62, 172.25, -54.5) mm, rotated rx -180 ry 0 rz 0.01 deg; joints [32.528, -38.785, 93.128, -142.11, 61.145, 160.401]
  MoveC 5813 to (-312.98, 176.27, -54.5) mm, rotated rx -180 ry 0 rz 0.01 deg; joints [32.718, -38.832, 93.22, -141.923, 61.249, 160.333] to (-311.32, 181.43, -54.5) mm, rotated rx 180 ry 0 rz 0.01 deg; joints [32.905, -38.769, 93.078, -141.697, 61.254, 160.179]
  MoveL 5814 to (-301.15, 283.24, -54.5) mm, rotated rx -180 ry 0 rz 0.01 deg; joints [36.05, -36.412, 87.899, -137.357, 60.339, 156.428]
  MoveC 5815 to (-302.02, 285.87, -54.5) mm, rotated rx -180 ry 0 rz 0.01 deg; joints [36.106, -36.299, 87.655, -137.248, 60.267, 156.297] to (-304.55, 287, -54.5) mm, rotated rx -180 ry 0 rz 0.01 deg; joints [36.086, -36.16, 87.36, -137.208, 60.143, 156.185]
  MoveL 5816 to (-347.73, 287, -54.5) mm, rotated rx -180 ry 0 rz 0.01 deg; joints [35.228, -34.313, 83.456, -137.275, 58.26, 155.029]
  MoveC 5817 to (-350.46, 285.87, -54.5) mm, rotated rx 180 ry 0 rz 0.01 deg; joints [35.144, -34.227, 83.276, -137.324, 58.154, 155.002] to (-351.58, 283.15, -54.5) mm, rotated rx -180 ry 0 rz 0.01 deg; joints [35.047, -34.26, 83.349, -137.443, 58.141, 155.089]
  MoveL 5818 to (-351.58, 249.25, -54.5) mm, rotated rx -180 ry 0 rz 0.01 deg; joints [34.1, -35.259, 85.51, -138.923, 58.598, 156.535]
  MoveC 5819 to (-352.65, 245.73, -54.5) mm, rotated rx 180 ry 0 rz 0.01 deg; joints [33.981, -35.314, 85.631, -139.077, 58.597, 156.653] to (-355.49, 243.39, -54.5) mm, rotated rx -180 ry 0 rz 0.01 deg; joints [33.86, -35.257, 85.514, -139.181, 58.502, 156.675]
  MoveC 5820 to (-358.33, 241.05, -54.5) mm, rotated rx -180 ry 0 rz 0.01 deg; joints [33.74, -35.199, 85.396, -139.285, 58.406, 156.697] to (-359.39, 237.53, -54.5) mm, rotated rx -180 ry 0 rz 0.01 deg; joints [33.62, -35.252, 85.514, -139.439, 58.405, 156.815]
  MoveL 5821 to (-359.39, 135.91, -54.5) mm, rotated rx 180 ry 0 rz 0.01 deg; joints [30.637, -37.911, 91.323, -143.824, 59.73, 160.779]
  MoveC 5822 to (-358.28, 134.09, -54.5) mm, rotated rx -180 ry 0 rz 0.01 deg; joints [30.602, -38.002, 91.519, -143.898, 59.804, 160.871] to (-356.15, 134.25, -54.5) mm, rotated rx 180 ry 0 rz 0.01 deg; joints [30.645, -38.088, 91.702, -143.885, 59.897, 160.913]
  MoveL 5823 to (-309.2, 167.97, -54.5) mm, rotated rx 180 ry 0 rz 0.01 deg; joints [32.541, -39.191, 94.002, -142.253, 61.52, 160.721]
  MoveC 5824 to (-305.56, 171.98, -54.5) mm, rotated rx -180 ry 0 rz 0.01 deg; joints [32.733, -39.237, 94.093, -142.064, 61.624, 160.654] to (-303.9, 177.14, -54.5) mm, rotated rx -180 ry 0 rz 0.01 deg; joints [32.92, -39.174, 93.952, -141.839, 61.627, 160.502]
  MoveL 5825 to (-292.52, 291.05, -54.5) mm, rotated rx -180 ry 0 rz 0.01 deg; joints [36.445, -36.537, 88.153, -136.995, 60.6, 156.322]
  MoveC 5826 to (-293.39, 293.68, -54.5) mm, rotated rx 180 ry 0 rz 0.01 deg; joints [36.5, -36.424, 87.908, -136.887, 60.528, 156.19] to (-295.92, 294.81, -54.5) mm, rotated rx 180 ry 0 rz 0.01 deg; joints [36.479, -36.286, 87.614, -136.848, 60.405, 156.079]
  MoveL 5827 to (-355.54, 294.81, -54.5) mm, rotated rx 180 ry 0 rz 0.01 deg; joints [35.291, -33.726, 82.208, -136.928, 57.804, 154.463]
  MoveC 5828 to (-358.27, 293.68, -54.5) mm, rotated rx 180 ry 0 rz 0.01 deg; joints [35.207, -33.639, 82.026, -136.975, 57.697, 154.434] to (-359.4, 290.96, -54.5) mm, rotated rx -180 ry 0 rz 0.01 deg; joints [35.111, -33.672, 82.101, -137.095, 57.684, 154.523]
  MoveL 5829 to (-359.39, 237.53, -54.5) mm, rotated rx -180 ry 0 rz 0.01 deg; joints [33.62, -35.252, 85.514, -139.439, 58.405, 156.815]
  MoveC 5830 to (-360.46, 234.01, -54.5) mm, rotated rx 180 ry 0 rz 0.01 deg; joints [33.5, -35.305, 85.631, -139.593, 58.404, 156.933] to (-363.3, 231.67, -54.5) mm, rotated rx -180 ry 0 rz 0.01 deg; joints [33.38, -35.247, 85.51, -139.697, 58.307, 156.954]
  MoveC 5831 to (-366.14, 229.33, -54.5) mm, rotated rx -180 ry 0 rz 0.01 deg; joints [33.26, -35.187, 85.389, -139.8, 58.21, 156.976] to (-367.2, 225.81, -54.5) mm, rotated rx 180 ry 0 rz 0.01 deg; joints [33.14, -35.239, 85.504, -139.954, 58.209, 157.093]
  MoveL 5832 to (-367.2, 120.69, -54.5) mm, rotated rx 180 ry 0 rz 0.01 deg; joints [30.035, -37.945, 91.42, -144.5, 59.572, 161.159]
  MoveC 5833 to (-366.09, 118.87, -54.5) mm, rotated rx 180 ry 0 rz 0.01 deg; joints [29.999, -38.035, 91.615, -144.575, 59.646, 161.25] to (-363.96, 119.03, -54.5) mm, rotated rx 180 ry 0 rz 0.01 deg; joints [30.042, -38.121, 91.799, -144.561, 59.74, 161.292]
  MoveL 5834 to (-301.78, 163.68, -54.5) mm, rotated rx 180 ry 0 rz 0.01 deg; joints [32.555, -39.592, 94.868, -142.392, 61.893, 161.037]
  MoveC 5835 to (-298.14, 167.7, -54.5) mm, rotated rx -180 ry 0 rz 0.01 deg; joints [32.747, -39.637, 94.959, -142.202, 61.996, 160.97] to (-296.48, 172.85, -54.5) mm, rotated rx -180 ry 0 rz 0.01 deg; joints [32.936, -39.576, 94.818, -141.976, 61.999, 160.819]
  MoveL 5836 to (-283.89, 298.86, -54.5) mm, rotated rx -180 ry 0 rz 0.01 deg; joints [36.84, -36.658, 88.397, -136.633, 60.859, 156.214]
  MoveC 5837 to (-284.76, 301.5, -54.5) mm, rotated rx -180 ry 0 rz 0.01 deg; joints [36.895, -36.544, 88.152, -136.525, 60.787, 156.082] to (-287.29, 302.62, -54.5) mm, rotated rx 180 ry 0 rz 0.01 deg; joints [36.873, -36.407, 87.86, -136.488, 60.665, 155.971]
  MoveL 5838 to (-363.35, 302.62, -54.5) mm, rotated rx 180 ry 0 rz 0.01 deg; joints [35.353, -33.13, 80.942, -136.571, 57.345, 153.884]
  MoveC 5839 to (-366.08, 301.49, -54.5) mm, rotated rx -180 ry 0 rz 0.01 deg; joints [35.27, -33.041, 80.757, -136.616, 57.237, 153.853] to (-367.21, 298.77, -54.5) mm, rotated rx 180 ry 0 rz 0.01 deg; joints [35.174, -33.075, 80.833, -136.736, 57.223, 153.943]
  MoveL 5840 to (-367.2, 225.81, -54.5) mm, rotated rx 180 ry 0 rz 0.01 deg; joints [33.14, -35.239, 85.504, -139.954, 58.209, 157.093]
  MoveC 5841 to (-368.27, 222.29, -54.5) mm, rotated rx -180 ry 0 rz 0.01 deg; joints [33.02, -35.29, 85.618, -140.108, 58.208, 157.21] to (-371.11, 219.96, -54.5) mm, rotated rx 180 ry 0 rz 0.01 deg; joints [32.9, -35.23, 85.494, -140.212, 58.11, 157.231]
  MoveC 5842 to (-373.95, 217.62, -54.5) mm, rotated rx -180 ry 0 rz 0.01 deg; joints [32.781, -35.17, 85.37, -140.315, 58.012, 157.252] to (-375.02, 214.1, -54.5) mm, rotated rx 180 ry 0 rz 0.01 deg; joints [32.66, -35.22, 85.481, -140.469, 58.01, 157.368]
  MoveL 5843 to (-375.01, 105.46, -54.5) mm, rotated rx 180 ry 0 rz 0.01 deg; joints [29.432, -37.969, 91.499, -145.175, 59.41, 161.536]
  MoveC 5844 to (-373.9, 103.64, -54.5) mm, rotated rx 180 ry 0 rz 0.01 deg; joints [29.395, -38.059, 91.693, -145.251, 59.483, 161.626] to (-371.77, 103.8, -54.5) mm, rotated rx -180 ry 0 rz 0.01 deg; joints [29.437, -38.146, 91.877, -145.238, 59.578, 161.667]
  MoveL 5845 to (-293.71, 159.86, -54.5) mm, rotated rx 180 ry 0 rz 0.01 deg; joints [32.595, -40.003, 95.757, -142.503, 62.286, 161.346]
  MoveC 5846 to (-290.57, 163.32, -54.5) mm, rotated rx 180 ry 0 rz 0.01 deg; joints [32.762, -40.042, 95.834, -142.338, 62.373, 161.289] to (-289.14, 167.78, -54.5) mm, rotated rx -180 ry 0 rz 0.01 deg; joints [32.926, -39.989, 95.714, -142.143, 62.376, 161.16]
  MoveL 5847 to (-275.47, 304.47, -54.5) mm, rotated rx 180 ry 0 rz 0.01 deg; joints [37.171, -36.831, 88.757, -136.361, 61.134, 156.191]
  MoveC 5848 to (-275.36, 305.06, -54.5) mm, rotated rx 180 ry 0 rz 0.01 deg; joints [37.19, -36.818, 88.728, -136.336, 61.131, 156.169] to (-275.24, 305.64, -54.5) mm, rotated rx -180 ry 0 rz 0.01 deg; joints [37.208, -36.806, 88.701, -136.311, 61.128, 156.148]
  MoveC 5849 to (-275.11, 306.23, -54.5) mm, rotated rx 180 ry 0 rz 0.01 deg; joints [37.227, -36.794, 88.674, -136.286, 61.126, 156.127] to (-275, 306.82, -54.5) mm, rotated rx 180 ry 0 rz 0.01 deg; joints [37.246, -36.78, 88.646, -136.261, 61.122, 156.105]
  MoveC 5850 to (-275.69, 309.33, -54.5) mm, rotated rx 180 ry 0 rz 0.01 deg; joints [37.301, -36.677, 88.423, -136.158, 61.06, 155.983] to (-278.05, 310.43, -54.5) mm, rotated rx 180 ry 0 rz 0.01 deg; joints [37.281, -36.549, 88.148, -136.122, 60.946, 155.877]
  MoveL 5851 to (-371.16, 310.43, -54.5) mm, rotated rx 180 ry 0 rz 0.01 deg; joints [35.414, -32.523, 79.655, -136.203, 56.881, 153.29]
  MoveC 5852 to (-373.89, 309.3, -54.5) mm, rotated rx 180 ry 0 rz 0.01 deg; joints [35.332, -32.433, 79.468, -136.247, 56.772, 153.258] to (-375.02, 306.58, -54.5) mm, rotated rx 180 ry 0 rz 0.01 deg; joints [35.236, -32.468, 79.546, -136.366, 56.758, 153.349]
  MoveL 5853 to (-375.02, 214.1, -54.5) mm, rotated rx 180 ry 0 rz 0.01 deg; joints [32.66, -35.22, 85.481, -140.469, 58.01, 157.368]
  MoveC 5854 to (-376.08, 210.58, -54.5) mm, rotated rx 180 ry 0 rz 0.01 deg; joints [32.539, -35.269, 85.592, -140.623, 58.008, 157.484] to (-378.92, 208.24, -54.5) mm, rotated rx 180 ry 0 rz 0.01 deg; joints [32.42, -35.208, 85.465, -140.726, 57.909, 157.505]
  MoveC 5855 to (-381.76, 205.9, -54.5) mm, rotated rx -180 ry 0 rz 0.01 deg; joints [32.301, -35.145, 85.337, -140.829, 57.81, 157.526] to (-382.83, 202.38, -54.5) mm, rotated rx 180 ry 0 rz 0.01 deg; joints [32.18, -35.194, 85.445, -140.983, 57.808, 157.641]
  MoveL 5856 to (-382.82, 90.24, -54.5) mm, rotated rx 180 ry 0 rz 0.01 deg; joints [28.829, -37.985, 91.558, -145.851, 59.243, 161.908]
  MoveC 5857 to (-381.71, 88.42, -54.5) mm, rotated rx -180 ry 0 rz 0.01 deg; joints [28.791, -38.074, 91.751, -145.926, 59.317, 161.997] to (-379.58, 88.57, -54.5) mm, rotated rx -180 ry 0 rz 0.01 deg; joints [28.833, -38.161, 91.937, -145.914, 59.412, 162.038]
  MoveL 5858 to (-287.93, 154.52, -54.5) mm, rotated rx -180 ry 0 rz 0.01 deg; joints [32.545, -40.357, 96.528, -142.688, 62.599, 161.657]
  MoveC 5859 to (-287.22, 155, -54.5) mm, rotated rx -180 ry 0 rz 0.01 deg; joints [32.574, -40.374, 96.562, -142.663, 62.623, 161.655] to (-286.48, 155.43, -54.5) mm, rotated rx -180 ry 0 rz 0.01 deg; joints [32.601, -40.392, 96.601, -142.64, 62.649, 161.655]
  MoveC 5860 to (-285.73, 155.83, -54.5) mm, rotated rx 180 ry 0 rz 0.01 deg; joints [32.628, -40.412, 96.642, -142.619, 62.675, 161.656] to (-284.97, 156.22, -54.5) mm, rotated rx 180 ry 0 rz 0.01 deg; joints [32.655, -40.431, 96.684, -142.597, 62.702, 161.658]
  MoveC 5861 to (-282.4, 158.7, -54.5) mm, rotated rx 180 ry 0 rz 0.01 deg; joints [32.782, -40.471, 96.766, -142.476, 62.778, 161.624] to (-281.57, 162.18, -54.5) mm, rotated rx 180 ry 0 rz 0.01 deg; joints [32.905, -40.42, 96.649, -142.326, 62.767, 161.518]
  MoveC 5862 to (-281.61, 163.09, -54.5) mm, rotated rx 180 ry 0 rz 0.01 deg; joints [32.932, -40.396, 96.596, -142.288, 62.754, 161.485] to (-281.65, 164, -54.5) mm, rotated rx -180 ry 0 rz 0.01 deg; joints [32.959, -40.372, 96.544, -142.25, 62.74, 161.452]
  MoveC 5863 to (-281.65, 164.92, -54.5) mm, rotated rx -180 ry 0 rz 0.01 deg; joints [32.987, -40.35, 96.494, -142.212, 62.728, 161.419] to (-281.59, 165.83, -54.5) mm, rotated rx 180 ry 0 rz 0.01 deg; joints [33.016, -40.33, 96.45, -142.174, 62.719, 161.388]
  MoveL 5864 to (-267.48, 306.1, -54.5) mm, rotated rx 180 ry 0 rz 0.01 deg; joints [37.384, -37.103, 89.332, -136.255, 61.444, 156.322]
  MoveC 5865 to (-267.02, 308.3, -54.5) mm, rotated rx -180 ry 0 rz 0.01 deg; joints [37.455, -37.056, 89.229, -136.161, 61.434, 156.242] to (-266.37, 310.46, -54.5) mm, rotated rx 180 ry 0 rz 0.01 deg; joints [37.528, -37.018, 89.143, -136.068, 61.431, 156.168]
  MoveC 5866 to (-265.68, 312.6, -54.5) mm, rotated rx -180 ry 0 rz 0.01 deg; joints [37.602, -36.981, 89.062, -135.976, 61.431, 156.096] to (-265.09, 314.77, -54.5) mm, rotated rx -180 ry 0 rz 0.01 deg; joints [37.675, -36.939, 88.971, -135.882, 61.426, 156.02]
  MoveC 5867 to (-265.6, 317.17, -54.5) mm, rotated rx -180 ry 0 rz 0.01 deg; joints [37.73, -36.847, 88.771, -135.785, 61.372, 155.907] to (-267.8, 318.24, -54.5) mm, rotated rx 180 ry 0 rz 0.01 deg; joints [37.712, -36.726, 88.514, -135.75, 61.267, 155.807]
  MoveL 5868 to (-378.98, 318.24, -54.5) mm, rotated rx 180 ry 0 rz 0.01 deg; joints [35.475, -31.904, 78.347, -135.824, 56.414, 152.68]
  MoveC 5869 to (-381.7, 317.11, -54.5) mm, rotated rx 180 ry 0 rz 0.01 deg; joints [35.392, -31.813, 78.157, -135.865, 56.303, 152.647] to (-382.83, 314.39, -54.5) mm, rotated rx 180 ry 0 rz 0.01 deg; joints [35.298, -31.849, 78.236, -135.985, 56.289, 152.739]
  MoveL 5870 to (-382.83, 202.38, -54.5) mm, rotated rx 180 ry 0 rz 0.01 deg; joints [32.18, -35.194, 85.445, -140.983, 57.808, 157.641]
  MoveC 5871 to (-383.89, 198.86, -54.5) mm, rotated rx 180 ry 0 rz 0.01 deg; joints [32.059, -35.242, 85.553, -141.137, 57.805, 157.756] to (-386.73, 196.52, -54.5) mm, rotated rx 180 ry 0 rz 0.01 deg; joints [31.94, -35.179, 85.422, -141.24, 57.706, 157.776]
  MoveC 5872 to (-389.57, 194.19, -54.5) mm, rotated rx 180 ry 0 rz 0.01 deg; joints [31.821, -35.115, 85.291, -141.342, 57.605, 157.797] to (-390.64, 190.66, -54.5) mm, rotated rx 180 ry 0 rz 0.01 deg; joints [31.7, -35.162, 85.396, -141.496, 57.602, 157.911]
  MoveL 5873 to (-390.63, 75.01, -54.5) mm, rotated rx 180 ry 0 rz 0.01 deg; joints [28.225, -37.992, 91.599, -146.526, 59.072, 162.277]
  MoveC 5874 to (-389.52, 73.19, -54.5) mm, rotated rx 180 ry 0 rz 0.01 deg; joints [28.187, -38.08, 91.791, -146.602, 59.146, 162.365] to (-387.39, 73.35, -54.5) mm, rotated rx 180 ry 0 rz 0.01 deg; joints [28.228, -38.168, 91.978, -146.59, 59.242, 162.406]
  MoveL 5875 to (-283.48, 148.33, -54.5) mm, rotated rx -180 ry 0 rz 0.01 deg; joints [32.442, -40.678, 97.228, -142.916, 62.867, 161.966]
  MoveC 5876 to (-281.5, 149.53, -54.5) mm, rotated rx 180 ry 0 rz 0.01 deg; joints [32.518, -40.725, 97.329, -142.852, 62.935, 161.965] to (-279.37, 150.44, -54.5) mm, rotated rx 180 ry 0 rz 0.01 deg; joints [32.588, -40.786, 97.458, -142.799, 63.013, 161.977]
  MoveC 5877 to (-277.16, 151.11, -54.5) mm, rotated rx 180 ry 0 rz 0.01 deg; joints [32.652, -40.855, 97.606, -142.755, 63.096, 161.999] to (-274.91, 151.65, -54.5) mm, rotated rx 180 ry 0 rz 0.01 deg; joints [32.713, -40.929, 97.763, -142.716, 63.183, 162.026]
  MoveC 5878 to (-272.87, 153.11, -54.5) mm, rotated rx 180 ry 0 rz 0.01 deg; joints [32.799, -40.972, 97.854, -142.64, 63.249, 162.016] to (-272.58, 155.6, -54.5) mm, rotated rx 180 ry 0 rz 0.01 deg; joints [32.881, -40.924, 97.745, -142.534, 63.229, 161.935]
  MoveC 5879 to (-273.04, 157.19, -54.5) mm, rotated rx 180 ry 0 rz 0.01 deg; joints [32.921, -40.868, 97.622, -142.472, 63.189, 161.87] to (-273.44, 158.8, -54.5) mm, rotated rx -180 ry 0 rz 0.01 deg; joints [32.962, -40.814, 97.504, -142.408, 63.152, 161.805]
  MoveC 5880 to (-273.75, 160.43, -54.5) mm, rotated rx 180 ry 0 rz 0.01 deg; joints [33.006, -40.763, 97.391, -142.343, 63.117, 161.742] to (-273.95, 162.08, -54.5) mm, rotated rx -180 ry 0 rz 0.01 deg; joints [33.053, -40.716, 97.287, -142.276, 63.088, 161.68]
  MoveC 5881 to (-274, 162.82, -54.5) mm, rotated rx -180 ry 0 rz 0.01 deg; joints [33.075, -40.696, 97.242, -142.245, 63.076, 161.652] to (-274.04, 163.57, -54.5) mm, rotated rx 180 ry 0 rz 0.01 deg; joints [33.097, -40.676, 97.198, -142.214, 63.064, 161.625]
  MoveC 5882 to (-274.05, 164.32, -54.5) mm, rotated rx 180 ry 0 rz 0.01 deg; joints [33.12, -40.658, 97.157, -142.183, 63.054, 161.598] to (-274.01, 165.07, -54.5) mm, rotated rx 180 ry 0 rz 0.01 deg; joints [33.143, -40.641, 97.121, -142.152, 63.046, 161.573]
  MoveL 5883 to (-259.86, 305.75, -54.5) mm, rotated rx -180 ry 0 rz 0.01 deg; joints [37.536, -37.416, 89.997, -136.231, 61.763, 156.523]
  MoveC 5884 to (-259.16, 308.54, -54.5) mm, rotated rx -180 ry 0 rz 0.01 deg; joints [37.629, -37.361, 89.876, -136.111, 61.754, 156.425] to (-258.32, 311.3, -54.5) mm, rotated rx 180 ry 0 rz 0.01 deg; joints [37.723, -37.312, 89.767, -135.992, 61.751, 156.331]
  MoveC 5885 to (-257.39, 314.03, -54.5) mm, rotated rx -180 ry 0 rz 0.01 deg; joints [37.818, -37.267, 89.668, -135.874, 61.752, 156.241] to (-256.38, 316.73, -54.5) mm, rotated rx -180 ry 0 rz 0.01 deg; joints [37.914, -37.226, 89.577, -135.756, 61.757, 156.153]
  MoveC 5886 to (-255.67, 318.3, -54.5) mm, rotated rx -180 ry 0 rz 0.01 deg; joints [37.973, -37.207, 89.534, -135.687, 61.765, 156.106] to (-254.78, 319.78, -54.5) mm, rotated rx 180 ry 0 rz 0.01 deg; joints [38.032, -37.198, 89.512, -135.621, 61.782, 156.066]
  MoveC 5887 to (-253.84, 321.22, -54.5) mm, rotated rx -180 ry 0 rz 0.01 deg; joints [38.092, -37.191, 89.496, -135.557, 61.8, 156.029] to (-252.96, 322.7, -54.5) mm, rotated rx -180 ry 0 rz 0.01 deg; joints [38.151, -37.181, 89.473, -135.491, 61.816, 155.989]
  MoveC 5888 to (-252.98, 324.94, -54.5) mm, rotated rx -180 ry 0 rz 0.01 deg; joints [38.213, -37.113, 89.324, -135.398, 61.785, 155.895] to (-254.92, 326.06, -54.5) mm, rotated rx 180 ry 0 rz 0.01 deg; joints [38.201, -37.002, 89.088, -135.362, 61.691, 155.8]
  MoveL 5889 to (-386.79, 326.05, -54.5) mm, rotated rx 180 ry 0 rz 0.01 deg; joints [35.534, -31.274, 77.016, -135.433, 55.942, 152.055]
  MoveC 5890 to (-389.51, 324.92, -54.5) mm, rotated rx -180 ry 0 rz 0.01 deg; joints [35.453, -31.181, 76.823, -135.472, 55.83, 152.019] to (-390.64, 322.2, -54.5) mm, rotated rx 180 ry 0 rz 0.01 deg; joints [35.359, -31.218, 76.904, -135.592, 55.816, 152.113]
  MoveL 5891 to (-390.64, 190.66, -54.5) mm, rotated rx -180 ry 0 rz 0.01 deg; joints [31.7, -35.162, 85.396, -141.496, 57.602, 157.911]
  MoveL 5892 to (-390.48, 190.06, -54.33) mm, rotated rx 180 ry 0 rz 0.01 deg; joints [31.685, -35.193, 85.448, -141.52, 57.612, 157.935]
  MoveL 5893 to (-390.19, 189.7, -53.87) mm, rotated rx 180 ry 0 rz 0.01 deg; joints [31.68, -35.237, 85.499, -141.529, 57.616, 157.944]
  MoveL 5894 to (-390.05, 189.6, -53.23) mm, rotated rx 180 ry 0 rz 0.01 deg; joints [31.679, -35.276, 85.522, -141.524, 57.604, 157.933]
  Set speed (500.0 mm/s)
  MoveL 5895 to (-390.05, 189.6, 11) mm, rotated rx 180 ry 0 rz 0.01 deg; joints [31.646, -38.157, 85.757, -140.459, 55.533, 155.956]
  Set speed (500.0 mm/s)
  MoveL 5896 to (-206.45, 109.97, 11) mm, rotated rx -180 ry 0 rz 0.01 deg; joints [32.751, -47.821, 105.6, -142.959, 63.949, 162.644]
  Set speed (500.0 mm/s)
  MoveL 5897 to (-206.45, 109.97, -32.73) mm, rotated rx 180 ry 0 rz 0.01 deg; joints [32.776, -45.55, 105.481, -143.539, 65.681, 164.057]
  Set speed (100.0 mm/s)
  MoveL 5898 to (-206.47, 109.81, -33.35) mm, rotated rx -180 ry 0 rz 0.01 deg; joints [32.771, -45.52, 105.485, -143.554, 65.707, 164.081]
  MoveL 5899 to (-206.5, 109.37, -33.82) mm, rotated rx -180 ry 0 rz 0.01 deg; joints [32.756, -45.504, 105.503, -143.578, 65.729, 164.109]
  MoveL 5900 to (-206.48, 108.75, -34) mm, rotated rx -180 ry 0 rz 0.01 deg; joints [32.736, -45.509, 105.534, -143.606, 65.745, 164.135]
  MoveL 5901 to (-202.46, 103.51, -34.24) mm, rotated rx -180 ry 0 rz 0.01 deg; joints [32.65, -45.757, 106.102, -143.782, 65.977, 164.381]
  MoveL 5902 to (-196.05, 105.1, -34.49) mm, rotated rx -180 ry 0 rz 0.01 deg; joints [32.837, -45.938, 106.515, -143.647, 66.219, 164.45]
  MoveL 5903 to (-194.93, 111.61, -34.73) mm, rotated rx 180 ry 0 rz 0.01 deg; joints [33.073, -45.82, 106.277, -143.368, 66.191, 164.269]
  MoveL 5904 to (-200.45, 115.24, -34.98) mm, rotated rx 180 ry 0 rz 0.01 deg; joints [33.074, -45.529, 105.671, -143.283, 65.939, 164.063]
  MoveL 5905 to (-205.99, 111.64, -35.22) mm, rotated rx -180 ry 0 rz 0.01 deg; joints [32.841, -45.398, 105.423, -143.496, 65.776, 164.089]
  MoveL 5906 to (-204.9, 105.12, -35.46) mm, rotated rx -180 ry 0 rz 0.01 deg; joints [32.652, -45.569, 105.828, -143.757, 65.909, 164.324]
  MoveL 5907 to (-198.5, 103.5, -35.71) mm, rotated rx -180 ry 0 rz 0.01 deg; joints [32.733, -45.821, 106.4, -143.755, 66.191, 164.496]
  MoveL 5908 to (-194.45, 108.72, -35.95) mm, rotated rx 180 ry 0 rz 0.01 deg; joints [32.99, -45.836, 106.451, -143.497, 66.294, 164.408]
  MoveL 5909 to (-197.61, 114.52, -36.2) mm, rotated rx -180 ry 0 rz 0.01 deg; joints [33.112, -45.582, 105.919, -143.296, 66.107, 164.174]
  MoveL 5910 to (-204.19, 113.95, -36.44) mm, rotated rx -180 ry 0 rz 0.01 deg; joints [32.955, -45.346, 105.44, -143.396, 65.865, 164.084]
  MoveL 5911 to (-206.31, 107.7, -36.68) mm, rotated rx 180 ry 0 rz 0.01 deg; joints [32.707, -45.397, 105.587, -143.68, 65.869, 164.255]
  MoveL 5912 to (-201.42, 103.25, -36.93) mm, rotated rx -180 ry 0 rz 0.01 deg; joints [32.664, -45.657, 106.182, -143.813, 66.127, 164.491]
  MoveL 5913 to (-195.39, 105.94, -37.17) mm, rotated rx -180 ry 0 rz 0.01 deg; joints [32.88, -45.799, 106.511, -143.637, 66.34, 164.518]
  MoveL 5914 to (-195.44, 112.55, -37.42) mm, rotated rx -180 ry 0 rz 0.01 deg; joints [33.094, -45.638, 106.178, -143.368, 66.264, 164.314]
  MoveL 5915 to (-201.51, 115.15, -37.66) mm, rotated rx 180 ry 0 rz 0.01 deg; joints [33.05, -45.351, 105.581, -143.332, 66.003, 164.131]
  MoveL 5916 to (-206.33, 110.63, -37.9) mm, rotated rx -180 ry 0 rz 0.01 deg; joints [32.803, -45.266, 105.434, -143.574, 65.879, 164.199]
  MoveL 5917 to (-204.12, 104.41, -38.15) mm, rotated rx -180 ry 0 rz 0.01 deg; joints [32.646, -45.47, 105.912, -143.81, 66.054, 164.444]
  MoveL 5918 to (-197.53, 103.94, -38.39) mm, rotated rx -180 ry 0 rz 0.01 deg; joints [32.769, -45.702, 106.44, -143.759, 66.329, 164.583]
  MoveL 5919 to (-194.46, 109.79, -38.64) mm, rotated rx 180 ry 0 rz 0.01 deg; joints [33.026, -45.669, 106.385, -143.485, 66.385, 164.458]
  MoveL 5920 to (-198.59, 114.94, -38.88) mm, rotated rx -180 ry 0 rz 0.01 deg; joints [33.106, -45.395, 105.81, -143.322, 66.167, 164.228]
  MoveL 5921 to (-204.97, 113.22, -39.12) mm, rotated rx -180 ry 0 rz 0.01 deg; joints [32.916, -45.193, 105.403, -143.467, 65.947, 164.177]
